// SIMATIC STEP 7 (V5.x) project kuphg_sepGsp2
// CPU: CPU 414-3 PN/DP
// station: P_ADR_BUS
// station: Hardware
// station: kuphg_sepGsp2
// program: S7 Program(2)

SYMBOL_TABLE
"db_Temp"	DB 1	DB 1
"db_BU"	DB 2	DB 2
"db_PIPE"	DB 3	DB 3
"db_Cmmn"	DB 4	DB 4
"idb_fb_Cnvt_Float1"	DB 5	FB 3
"idb_fb_Cnvt_Com"	DB 6	FB 2
"db_MsgCrane"	DB 7	DB 7
"idb_fb_QueueEx"	DB 8	FB 4
"idb_fb_DownloadSnd"	DB 9	FB 10
"idb_fb_Put"	DB 10	FB 6
"idb_fb_Get"	DB 11	FB 7
"idb_fb_Solver"	DB 12	FB 8
"idb_fb_DataFill"	DB 13	FB 9
"db_FIFO"	DB 14	DB 14
"idb_fb_Restart"	DB 15	FB 11
"idb_fb_Scada_Snd"	DB 16	FB 12
"db_MsgInd"	DB 17	DB 17
"idb_fb_Cnvt_Float2"	DB 18	FB 5
"idb_fb_Cnvt_Byte1"	DB 19	FB 14
"idb_fb_Cnvt_Bool1"	DB 20	FB 15
"idb_fb_Cnvt_Bool2"	DB 21	FB 16
"idb_fb_confDown"	DB 22	FB 13
"idb_fb_Snd_Rcv_CP00"	DB 25	FB 18
"idb_fb_Snd_Rcv_CP01"	DB 26	FB 19
"idb_FB_Test"	DB 30	FB 1
"db_MsgCru"	DB 36	DB 36
"idb_fb_StatusRcv"	DB 38	FB 26
"db_MsgPress"	DB 39	DB 39
"db_MsgPPress"	DB 40	DB 40
"db_MsgTemp"	DB 41	DB 41
"db_MsgFlow"	DB 42	DB 42
"db_MsgWorkReg"	DB 43	DB 43
"db_MsgPipeMsg"	DB 44	DB 44
"db_MsgOper"	DB 45	DB 45
"db_MsgInfo"	DB 46	DB 46
"db_MsgOther"	DB 47	DB 47
"idb_snd00"	DB 112	SFB 12
"idb_rcv00"	DB 113	SFB 13
"idb_snd01"	DB 122	SFB 12
"idb_rcv01"	DB 123	SFB 13
"idb_sts00"	DB 201	SFB 22
"idb_sts01"	DB 202	SFB 22
"DbDeb1"	DB 220	DB 220
"DbInfo"	DB 221	DB 221
"DbSensBool"	DB 222	DB 222
"DbSensAI"	DB 223	DB 223
"DbKranPpuAdr"	DB 224	DB 224
"DbKranPpu"	DB 225	DB 225
"DbSepBu"	DB 226	DB 226
"DbSipValve"	DB 227	DB 227
"DbFlowData"	DB 228	DB 228
"DbBitMess"	DB 229	DB 229
"DbControl"	DB 230	DB 230
"DbFlowControl"	DB 231	DB 231
"DbSepBlow"	DB 232	DB 232
"DbCaution"	DB 233	DB 233
"DbEnum"	DB 234	DB 234
"DbSipValveDeb"	DB 248	DB 248
"DbKranPpuDeb"	DB 249	DB 249
"idb_fb_ParScan"	DB 251	FB 251
"idb_fb_KranPpu"	DB 252	FB 252
"idb_fb_Watch"	DB 253	FB 253
"idb_fb_ExecCmd"	DB 254	FB 254
"idb_fb_SipValve"	DB 255	FB 255
"idb_fb_Flow"	DB 256	FB 256
"db_BSEND"	DB 292	SFB 12
"db_BRCV"	DB 293	SFB 13
"DbCpBufSend"	DB 294	DB 294
"DbCpBufRcv"	DB 295	DB 295
"fb_Test"	FB 1	FB 1
"fb_Cnvt_Com"	FB 2	FB 2
"fb_Cnvt_Float1"	FB 3	FB 3
"fb_QueueEx"	FB 4	FB 4
"fb_Cnvt_Float2"	FB 5	FB 5
"fb_Put"	FB 6	FB 6
"fb_Get"	FB 7	FB 7
"fb_Solver"	FB 8	FB 8
"fb_DataFill"	FB 9	FB 9
"fb_DownloadSnd"	FB 10	FB 10
"fb_Restart"	FB 11	FB 11
"fb_Scada_Snd"	FB 12	FB 12
"fb_confDown"	FB 13	FB 13
"fb_Cnvt_Byte1"	FB 14	FB 14
"fb_Cnvt_Bool1"	FB 15	FB 15
"fb_Cnvt_Bool2"	FB 16	FB 16
"fb_Snd_Rcv_CP00"	FB 18	FB 18
"fb_Snd_Rcv_CP01"	FB 19	FB 19
"fb_StatusRcv"	FB 26	FB 26
"fb_ParScan"	FB 251	FB 251
"fb_KranPpu"	FB 252	FB 252
"fb_Watch"	FB 253	FB 253
"fb_ExecCmd"	FB 254	FB 254
"fb_SipValve"	FB 255	FB 255
"fb_Flow"	FB 256	FB 256
"fc_is_empty"	FC 1	FC 1
"CONCAT"	FC 2	FC 2	// Concatenate  String
"fc_MsgSet"	FC 5	FC 5
"fc_MsgReset"	FC 6	FC 6
"fc_MsgHandlerCycle"	FC 7	FC 7
"DT to TOD"	FC 8	FC 8	// DT to TOD
"fc_MsgIsSet"	FC 9	FC 9
"fc_MsgHandlerCrane"	FC 10	FC 10
"I_STRNG"	FC 16	FC 16	// Integer to String
"LEN"	FC 21	FC 21	// Length of String
"MID"	FC 26	FC 26	// Middle Part of String
"RIGHT"	FC 32	FC 32	// Right Part of String
"S5TI_TIM"	FC 33	FC 33	// S5 Time to IEC Time
"SB_DT_DT"	FC 34	FC 34	// Subtract DT - DT
"SB_DT_TM"	FC 35	FC 35	// Subtract DT Time
"TIM_S5TI"	FC 40	FC 40	// IEC Time to S5 Time
"SCALE"	FC 105	FC 105	// Scaling Values
"UNSCALE"	FC 106	FC 106	// Unscaling Values
"FcSetBit"	FC 251	FC 251
"FcBcdByteToInt"	FC 252	FC 252
"FcIntToDt"	FC 253	FC 253
"FcDtToInt"	FC 254	FC 254
"FcDtIntToStr"	FC 255	FC 255
"FcCalcFlow"	FC 256	FC 256
"FcSetCaution"	FC 257	FC 257
"FcPlayCaution"	FC 258	FC 258
"fc_CRC16"	FC 1002	FC 1002	// у Чернова был Fc2 - заменено 20.05.2014
"obMain"	OB 1	OB 1
"obCyclicCalcFlow"	OB 32	OB 32
"obErrRunTime"	OB 80	OB 80
"obRestart"	OB 100	OB 100
"BSEND"	SFB 12	SFB 12	// Sending Segmented Data
"BRCV"	SFB 13	SFB 13	// Receiving Segmented Data
"STATUS"	SFB 22	SFB 22	// Query the Status of a Remote Partner
"SET_CLK"	SFC 0	SFC 0	// Set System Clock
"READ_CLK"	SFC 1	SFC 1	// Read System Clock
"ALARM_SQ"	SFC 17	SFC 17	// Generate Block-Related Messages with Acknowledgment
"ALARM_S"	SFC 18	SFC 18	// Generate Permanently Acknowledged Block-Related Messages
"ALARM_SC"	SFC 19	SFC 19	// Query the Acknowledgment Status of the last ALARM_SQ Entering State Message
"udt_Pipe"	UDT 1	UDT 1
"udt_Pipe_snd"	UDT 4	UDT 4
"udt_Snd"	UDT 5	UDT 5
"udt_Rcv"	UDT 6	UDT 6
"TAdrIOSignal"	UDT 201	UDT 201
"TSignalBool"	UDT 202	UDT 202
"TSignalAI"	UDT 203	UDT 203
"TKranPpu"	UDT 204	UDT 204
"TSepBuParam"	UDT 206	UDT 206
"TSipValve"	UDT 207	UDT 207
"TFlowData"	UDT 208	UDT 208
"TDateTimeBcd"	UDT 209	UDT 209
"TDateTimeInt"	UDT 210	UDT 210
"TSepBlow"	UDT 211	UDT 211
"TCaution"	UDT 212	UDT 212
"TSipValveDeb"	UDT 248	UDT 248
"TKranPpuDeb"	UDT 259	UDT 259
"Vat_Deb_Calc"	VAT 1	
"Vat_AI16_slot10_Piw"	VAT 2	
"Vat_AO8_slot11"	VAT 3	
"Vat_KrPpu_Tmp"	VAT 4	
"Vat_Zagaz"	VAT 5	
"Vat_KrPpu_01_All"	VAT 6	
"Vat_Timer"	VAT 7	
"Vat_DI_09-13zagaz"	VAT 8	
"Vat_Bu_Cfg"	VAT 9	
"Vat_DbSepBu"	VAT 10	
"Vat_Timer_v2"	VAT 11	
"Vat_KlapanSP"	VAT 12	
"Vat_TestBU"	VAT 13	
"vt_dwnld"	VAT 14	
"vt_Message"	VAT 15	
"vt_messtest"	VAT 16	
"vt_msg"	VAT 17	
"vt_Pipe_R0"	VAT 18	
"vt_Pipe_R1"	VAT 19	
"vt_Pipe_R12"	VAT 20	
"vt_Pipe_R6"	VAT 21	
"vt_Pipe_W"	VAT 22	
"vt_queue_ex"	VAT 23	
"vt_snd_rcv"	VAT 24	
"vt_test"	VAT 25	
"Vat_KrPpu_Emul_Si1"	VAT 26	
"Vat_KrPpu_01_Timers"	VAT 27	
"Vat_SensAI_15_Sp_Level"	VAT 28	
"Vat_KrPpu_HandPush"	VAT 29	
"Vat_SensAI_14_Sp_Rashod"	VAT 30	
"Vat_SipValve_3_SP"	VAT 31	
"Vat_KrPpu_All_State_ok"	VAT 32	
"Vat_SipValve_1_Si1"	VAT 33	
"Vat_SipValve_Time"	VAT 34	
"Vat_SipValve_2_Si2"	VAT 35	
"Vat_SipValve_4-5"	VAT 36	
"Vat_Mess"	VAT 37	
"Vat_Emul_Ai_KrPpu_SipVal"	VAT 38	
"Vat_FlowData_0"	VAT 39	
"Vat_FlowControl"	VAT 40	
"Vat_FlowData_1_Gaz_Si1"	VAT 41	
"Vat_ZagazUpr"	VAT 42	
"Vat_BcdDateTime"	VAT 43	
"Vat_FlowData_3_Sp"	VAT 44	
"Vat_BcdDateTime_2"	VAT 45	
"Vat_SensBool_Zagaz"	VAT 46	
"Vat_SensBool2"	VAT 47	
"Vat_SensAI_mA_All"	VAT 48	
"Vat_FlowCalcW"	VAT 49	
"Vat_BU_Uou_KK1"	VAT 50	
"Vat_SensAI_00"	VAT 51	
"Vat_FlowCalcW_1_Si1"	VAT 52	
"Vat_SipValve_4-5a"	VAT 53	
"Vat_FlowCalcW_3_Sp1+"	VAT 54	
"Vat_Caution_tStamp"	VAT 55	
END_SYMBOL_TABLE

TYPE "udt_Pipe"	// UDT 1
VERSION : 0.0
  STRUCT
   CP : INT ;
   PORT : INT ;
   BU : INT ;
   ADDR : BYTE ;	//краны 1,8,11 состояния
   Crane : ARRAY  [0 .. 2 ] OF STRUCT
    Inv : BOOL ;
    RMCntr : BOOL ;
    RComm_Fault : BOOL ;
    RCntr_State : BYTE ;
    RState : BYTE ;
    RCntr_Open : BYTE ;
    RCntr_Close : BYTE ;
    RHw_Error : BYTE ;	//CntrEnableOpen  :BOOL:=0; //0 - нет доступа
//CntrEnableClose  :BOOL:=0; //0 - не
    NeisprUpr : BOOL ;	//0 - неисправность отсутствует
   END_STRUCT ;	//КРУ
   KRU : STRUCT
    Inv : BOOL ;
    RComm_Fault : BOOL ;
    RHw_Fault : BOOL ;
    RCntr_Curr : BOOL ;
    ROpen_Fault : BOOL ;
    RClose_Fault : BOOL ;
    RCntr_Switch : BOOL ;
    RCntr_State : BYTE ;
    RPos_Drv : BYTE ;
    RCntr_Open : BYTE ;
    RCntr_Close : BYTE ;
    RCntr_Pow : BYTE ;
    RCal_Pos_Drv : REAL ;
    RMContr : REAL ;
    RACntr : REAL ;
    RCurr : REAL ;
    RP_PID : REAL ;
    RI_PID : REAL ;
    RD_PID : REAL ;
    CntrEnable : BOOL ;	//0 - нет доступа
    NeisprNoUpr : BOOL ;	//0 - неисправность отсутствует
    NeisprUpr : BOOL ;	//0 - неисправность отсутствует
   END_STRUCT ;
   Press : STRUCT
    Inv : BOOL ;
    RWarnNE : BOOL ;
    RBigNE : BOOL ;
    RWr : BOOL ;
    RA : BYTE ;
    RF : BYTE ;
    RVal : REAL ;
    RUpThres : REAL ;
    RDnThres : REAL ;
    RUpYellow : REAL ;
    RDnYellow : REAL ;
    RUpRed : REAL ;
    RDnRed : REAL ;
    Delta : INT ;
    Zones : INT ;
   END_STRUCT ;
   PPress : STRUCT
    Inv : BOOL ;
    RWr : BOOL ;
    RA : BYTE ;
    RF : BYTE ;
    RVal : REAL ;
    RUpThres : REAL ;
    RDnThres : REAL ;
    RUpYellow : REAL ;
    RDnYellow : REAL ;
    RUpRed : REAL ;
    RDnRed : REAL ;
    Delta : INT ;
    Zones : INT ;
   END_STRUCT ;
   Temp : STRUCT
    Inv : BOOL ;
    RWr : BOOL ;
    RA : BYTE ;
    RF : BYTE ;
    RVal : REAL ;
    RUpThres : REAL ;
    RDnThres : REAL ;
    RUpYellow : REAL ;
    RDnYellow : REAL ;
    RUpRed : REAL ;
    RDnRed : REAL ;
    Delta : INT ;
    Zones : INT ;
   END_STRUCT ;
   POST : STRUCT
    RReq : BOOL ;
    RVal : BOOL ;
   END_STRUCT ;
   FLOW : STRUCT
    Inv : BOOL ;
    RSwitch : BOOL ;
    RWr : BOOL ;
    RFault : BOOL ;
    RVal : REAL ;
    RUst : REAL ;
    RDens : REAL ;
    RDiamDiaf : REAL ;
    RDiamIT : REAL ;
    REqvSh : REAL ;
    RPressBar : REAL ;
    RCo2 : REAL ;
    RNitro : REAL ;
    RRad : REAL ;
    RCnt : REAL ;
    RFlowHour : REAL ;
    RFlowDay : REAL ;
    bSetpoint : BOOL ;
    bSetCalc : BOOL ;
    bSetHBD : BOOL ;
    bSetDBD : BOOL ;
    currHcalc : REAL ;
    prevHcalc : REAL ;
    currDcalc : REAL ;
    prevDcalc : REAL ;
    deltaFlow : REAL ;
    RiseFlow : REAL ;
   END_STRUCT ;
   WrkRegim : STRUCT
    RSwRegWrk : BOOL ;
    RGRP : BOOL ;
    RCntrReg : BYTE ;
    RRegWrk : BYTE ;
   END_STRUCT ;
   PipeMess : STRUCT
    RAlarmRed : BOOL ;
    RFaultTehn : BOOL ;
    RFaultCntr : BOOL ;
    RFaultHW : BOOL ;
    RFaultInt : BOOL ;
    RPermAlarm : BOOL ;
    RRstIntFault : BOOL ;
    RRepair : BOOL ;
    RGasNotBleed : BOOL ;
    RPipeGas : BOOL ;
   END_STRUCT ;
   Times : STRUCT
    RTime : ARRAY  [0 .. 10 ] OF BYTE ;
    RYear : INT ;
    RMonth : INT ;
    RDay : INT ;
    RDay_of_Week : INT ;
    RHour : INT ;
    RMinute : INT ;
    RSecond : INT ;
    RMSecond : INT ;
   END_STRUCT ;
   Ind : INT ;
   Invalid : BOOL ;
   CntrEnable : BOOL ;
   PipeWrkRegim : INT ;
   PipeSeason : INT ;
   cntrIOCranes : BOOL ;
   cntrCCrane : BOOL ;
   inCcIOCranes : BOOL ;
   inCcCCrane : BOOL ;
   inPmaxEkm : BOOL ;
   inPminEkm : BOOL ;
   cntrLedCCraneOP : BOOL ;
   inCCraneOP : BOOL ;
   inCcPmaxEkm : BOOL ;
   inCcPminEkm : BOOL ;
   bAlarmStopWinCC : BOOL ;
  END_STRUCT ;	
END_TYPE

TYPE "udt_Pipe_snd"	// UDT 4
VERSION : 0.0
  STRUCT 	//краны 1,8,11
   Crane : ARRAY  [0 .. 2 ] OF STRUCT
    WMCntr : BOOL ;
   END_STRUCT ;	//КРУ
   KRU : STRUCT
    WCntr_Switch : BOOL ;
    WMContr : REAL ;
    WP_PID : REAL ;
    WI_PID : REAL ;
    WD_PID : REAL ;
   END_STRUCT ;
   Press : STRUCT
    WWr : BOOL ;
    WUpThres : REAL ;
    WDnThres : REAL ;
    WUpYellow : REAL ;
    WDnYellow : REAL ;
    WUpRed : REAL ;
    WDnRed : REAL ;
   END_STRUCT ;
   PPress : STRUCT
    WWr : BOOL ;
    WUpThres : REAL ;
    WDnThres : REAL ;
    WUpYellow : REAL ;
    WDnYellow : REAL ;
    WUpRed : REAL ;
    WDnRed : REAL ;
   END_STRUCT ;
   Temp : STRUCT
    WWr : BOOL ;
    WUpThres : REAL ;
    WDnThres : REAL ;
    WUpYellow : REAL ;
    WDnYellow : REAL ;
    WUpRed : REAL ;
    WDnRed : REAL ;
   END_STRUCT ;
   POST : STRUCT
    WVal : BOOL ;
   END_STRUCT ;
   FLOW : STRUCT
    WSwitch : BOOL ;
    WWr : BOOL ;
    WUst : REAL ;
    WDens : REAL ;
    WDiamDiaf : REAL ;
    WDiamIT : REAL ;
    WEqvSh : REAL ;
    WPressBar : REAL ;
    WCo2 : REAL ;
    WNitro : REAL ;
    WRad : REAL ;
   END_STRUCT ;
   WrkRegim : STRUCT
    WSwRegWrk : BOOL ;
    WGRP : BOOL ;
    WCntrReg : BYTE ;
   END_STRUCT ;
   PipeMess : STRUCT
    WPermAlarm : BOOL ;
    WRstIntFault : BOOL ;
   END_STRUCT ;
   Times : STRUCT
    WTime : ARRAY  [0 .. 10 ] OF BYTE ;
    WYear : INT ;
    WMonth : INT ;
    WDay : INT ;
    WDay_of_Week : INT ;
    WHour : INT ;
    WMinute : INT ;
    WSecond : INT ;
    WMSecond : INT ;
   END_STRUCT ;
  END_STRUCT ;	
END_TYPE

TYPE "udt_Snd"	// UDT 5
VERSION : 0.0
  STRUCT
   adress : BYTE ;
   funct : BYTE ;
   Reg : WORD ;
   Ndata : INT ;
   Data : ARRAY  [0 .. 126 ] OF WORD ;
   Lenght : WORD ;
   Cmd : INT ;	// 0-опрос, 1-команда, 2-загрузка
   Pipe_N : INT ;
   Obj_N : INT ;
   Par_N : INT ;
   Bit : INT ;
  END_STRUCT ;	
END_TYPE

TYPE "udt_Rcv"	// UDT 6
VERSION : 0.0
  STRUCT
   rcv : ARRAY  [0 .. 126 ] OF WORD ;
   Ready : BOOL ;
   Invalid : BOOL ;
  END_STRUCT ;	
END_TYPE

TYPE "TAdrIOSignal"	// UDT 201
VERSION : 0.0
  STRUCT
   adr1 : INT ;
   adr2 : INT ;
  END_STRUCT ;	
END_TYPE

TYPE "TSignalBool"	// UDT 202
VERSION : 0.0
  STRUCT
   adr1 : INT ;
   adr2 : INT ;
   Value : BOOL ;
  END_STRUCT ;	
END_TYPE

TYPE "TSignalAI"	// UDT 203
VERSION : 0.0
  STRUCT
   adrPIW : INT ;	//адрес "слова" в PIW[] для вычисления значения датчика на AI-входе
   ValueIn : INT ;	//пре-обработанное цифровое значение датчика
   Value_mA : REAL ;	//токовое значение датчика (в мА)
   tStamp : DATE_AND_TIME ;	//метка времени в момент успешной обработки значения AI-датчика
   Value : REAL ;	//значение датчиков в момент tStamp (напр. +25.7 градС)
   Value_Subst : REAL ;	//+подстановочное значение
   SubstIncrement : REAL ;	//+ежецикличное приращение для подстановочного значения (меняет знак)
   lblErr : INT ;	//Признак ошибки:0-нет\1-отриц. переполн(<3.8мА)\2-переполн(>20.2мА)\3-обрыв
   lblBound : INT ;	//Признак наруш. границ:-1-неопр\0-Норма\1-LoLo\2-Lo\3-Hi\4-HiHi\>4-ошЗадГраниц
   lblModeSubst : BOOL ;	//+метка активации режима "подстановка значения": 1- "подстановка" \0-нет
   lblModeRepair : BOOL ;	//+метка активации режима "датчик в ремонте" : 1- "в ремонте" \0-нет
   lblSubstCalc : BOOL ;	//+метка активации "простого" пересчёта Value_Subst: 1- пересчитывать \0-нет
   lblSubstCalcBlow : BOOL ;	//+метка активации пересчёта Value_Subst с учетом продувок : 1- да\0-нет
   BoundLoLo : REAL ;	//нижняя аварийная граница
   BoundLo : REAL ;	//нижняя предупредительная граница
   BoundHi : REAL ;	//верхняя предупредительная граница
   BoundHiHi : REAL ;	//верхняя аварийная граница
   LoMeasure : REAL ;	//нижний предел измерения в физич. единицах (напр. -50 градС)
   HiMeasure : REAL ;	//верхний предел измерения в физич. единицах(напр. +100 градС)
   LoMeasure_mA : REAL ;	//нижний предел измерения,мА (const 4 мА для датчиков [4-20]мА)
   HiMeasure_mA : REAL ;	//верхний предел измерения,мА (const 20 мА для датчиков [4-20]мА)
   LoWorkRange_mA : REAL ;	//нижний рабочий предел измерения,мА (напр. 3.8 мА для датчиков [4-20]мА)
   HiWorkRange_mA : REAL ;	//верхний рабочий предел измерения,мА (напр. 20.2 мА для датчиков [4-20]мА)
   HmiBoundLoLo : REAL ;	//дублирующий пакет уставок для независимой корректировки на ВУ
   HmiBoundLo : REAL ;
   HmiBoundHi : REAL ;
   HmiBoundHiHi : REAL ;
   HmiLoMeasure : REAL ;
   HmiHiMeasure : REAL ;
   HmiLoWorkRange_mA : REAL ;
   HmiHiWorkRange_mA : REAL ;
   HmiSyncRange : INT ;	//синхр-ция знач. уставок ПЛК и ВУ:0-не проводить\1-синхрПЛК=>ВУ\2-синхрВУ=>ПЛК
   HmiSensAiDefect : BOOL ;	// Признак ошибочных показаний датчика для ВУ : 0 - правильные \ 1 - ошибочные
  END_STRUCT ;	
END_TYPE

TYPE "TKranPpu"	// UDT 204
VERSION : 0.0
  STRUCT
   KrClose : BOOL ;	//значение DI-сигнала крана ЭППУ "закрыт" (концевик закрытия)
   KrOpen : BOOL ;	//значение DI-сигнала крана ЭППУ "открыт" (концевик открытия)
   CC_Close : BOOL ;	//значение DI-сигнала крана ЭППУ "Целостность Цепи закрытия" :1 - естьЦЦ\0-нет
   CC_Open : BOOL ;	//значение DI-сигнала крана ЭППУ "Целостность Цепи открытия" :1 - естьЦЦ\0-нет
   KrToCloseR : BOOL ;	//значение DO-сигнала крана ЭППУ "закрыть" (чтение состояния)
   KrToCloseW : BOOL ;	//значение DO-сигнала "закрыть" (вычисляется за цикл и назначается в Q[x,5])
   KrToOpenR : BOOL ;	//значение DO-сигнала крана ЭППУ "открыть" (чтение состояния)
   KrToOpenW : BOOL ;	//значение DO-сигнала "открыть" (вычисляется за цикл и назначается в Q[x,5])
   KrToCloseW_HandPush : BOOL ;	//значение DO-сигнала "закрыть" (назначается в Q[x,5] при HandPush=true)
   KrToOpenW_HandPush : BOOL ;	//значение DO-сигнала "открыть" (назначается в Q[x,6] при HandPush=true)
   KrClose_NotSancMove : BOOL ;	//метка : 1- начало несанкцинир. закрытия крана с площадки \ 0- нет)
   KrOpen_NotSancMove : BOOL ;	//метка : 1- начало несанкцинир. открытия крана с площадки \ 0- нет)
   KrClose_PrevVal : BOOL ;	//предыдущее значение DI-сигнала крана ЭППУ "закрыт" (концевик закрытия)
   KrClose_Ev01 : BOOL ;	//флаг события "концевик закрытия замкнулся" (0->1) : 1- да \ 0- нет)
   KrClose_Ev10 : BOOL ;	//флаг события "концевик закрытия разомкнулся" (1->0) : 1- да \ 0- нет)
   KrOpen_PrevVal : BOOL ;	//предыдущее значение DI-сигнала крана ЭППУ "открыт" (концевик открытия)
   KrOpen_Ev01 : BOOL ;	//флаг события "концевик открытия замкнулся" (0->1) : 1- да \ 0- нет)
   KrOpen_Ev10 : BOOL ;	//флаг события "концевик открытия разомкнулся" (1->0) : 1- да \ 0- нет)
   TmOperKr_NO : INT ;	//номер таймера (используютя глобально) - инициализируется
   TmOperKr_TV : S5TIME ;	//величина таймера (длительность) - назначается взавис. от шага операции
   TmOperKr_Q : BOOL ;	//состояние таймера (для таймера типа s_odts : 1 - время отсчитано)
   TmStrag_Value : S5TIME ;	//время на страгивани крана
   TmFullClose_Value : S5TIME ;	//время на полное закрытие крана
   TmFullOpen_Value : S5TIME ;	//время на полное открытие крана
   TmDogim_Value : S5TIME ;	//время на дожим крана  //s5t#20ms
   HmiTmStrag_Value : DINT ;	//время на страгивани крана - для ВУ тип dInt
   HmiTmFullClose_Value : DINT ;	//время на полное закрытие крана - для ВУ тип dInt
   HmiTmFullOpen_Value : DINT ;	//время на полное открытие крана - для ВУ тип dInt
   HmiTmDogim_Value : DINT ;	//время на дожим крана  //s5t#20ms - для ВУ тип dInt
   State : INT ;	//сост-е крана:0-неопред.\1-закрыт\2-открыт\3-закрывается\4-открывается\5-неиспр
   StateByClOp : INT ;	//сост. крана по концевикам : 1-закрыт\2-открыт\3-ClOp00 (разомкнуты)\4-ClOp11
   CmdKrPpu : INT ;	//команда для крана : 0-нет\1-закрыть (с ВУ) \ 2-открыть (с ВУ)\..
   CmdKrPpuModeExec : INT ;	//режим исп.команды: 0-норм.\1-прин.прерыв.\2-прин.исп\3-экстренное исп.
   CmdKrPpu_Next : INT ;	//следующая команда для крана : 0-нет\1-закрыть (с ВУ) \ 2-открыть (с ВУ)\..
   CmdKrPpuModeExec_Next : INT ;	//режим исп.след.команды: 0-норм.\1-прин.прерыв.\2-прин.исп\3-экстренное исп.
   CmdKrPpuLegal : BOOL ;	//непротиворечивость команды : 0-нельзя исполнять\1-можно исполнять
   CmdKrPpuHandPush : BOOL ;	//ручное директивное управленне : 0-выключено\1-включено
   Oper : INT ;	//вып-яемая операция с краном : 0 - нет операций (стоит)\1-закрыть\2-открыть
   OperStep : INT ;	//шаг вып-яемой операции:0-нет\ 1Х-закрытие(11страг\12fullOpen\13дожим)\ 2Х-откр.
   OperErrorLbl : BOOL ;	//наличие ошибки при выполнении операции с краном : 0 - нет \ 1 - есть
   OperErrorNum : INT ;	//номер ошибки при выполнении операции с краном : 0 - нет ошибок \ 1 ..
   HmiErrCC_Close : BOOL ;	//метка : 1- нарушена ц.ц. на закрытие \ 0- нет
   HmiErrCC_Open : BOOL ;	//метка : 1- нарушена ц.ц. на открытие \ 0- нет
   HmiErrClOp00 : BOOL ;	//метка : 1- оба концевика в 0 (разомкнуты) \ 0- нет (ClOp - Close-Open)
   HmiErrClOp11 : BOOL ;	//метка : 1- оба концевика в 1 (замкнуты) \ 0- нет
   HmiErrMessConfirm : BOOL ;	//метка : 1- не квитированы сообщения \ 0- нет
   HmiSyncTimers : INT ;	//синхр-ция знач. таймеров ПЛК и ВУ:0-не проводить\1-синхрПЛК=>ВУ\2-синхрВУ=>ПЛК
   KrDefectFatal : BOOL ;	//фатальная неисправность крана - управление невозможно
   KrDefectNote : BOOL ;	//предупр. неисправность крана, при которой управление возможно
   HmiKrEnableToClose : BOOL ;	//доступность крана для закрытия с ВУ : 0-не доступен \ 1 - доступен
   HmiKrEnableToOpen : BOOL ;	//доступность крана для открытия с ВУ : 0-не доступен \ 1 - доступен
   HmiKrToClose : BOOL ;	//факт подачи команды на закрытие крана с ВУ : 0- не подана \ 1 - подана
   HmiKrToOpen : BOOL ;	//факт подачи команды на открытие крана с ВУ : 0- не подана \ 1 - подана
   isBan_AutoControl : BOOL ;	//флаг запрета автоматического управления краном: 0-нет запрета\ 1- запрещено
   isBan_HandControl : BOOL ;	//флаг запрета ручного управления краном: 0-нет запрета\ 1- запрещено
   reasonBan_AutoControl : INT ;	//причина запрета автоматического управления краном (RBC_ из DbEnum)
   reasonBan_HandControl : INT ;	//причина запрета ручного управления краном (RBC_ из DbEnum)
  END_STRUCT ;	
END_TYPE

TYPE "TSepBuParam"	// UDT 206
VERSION : 0.0
  STRUCT
   addr : BYTE ;	// дрес блока управления в HEX (из db_BU)
   vDbBu_Pipe0 : INT ;	// номер 1-й нитки для шлейфа 57 БУ (номер эл-та в db_Pipe (начинается с 0)
   vDbBu_Pipe1 : INT ;	// номер 2-й нитки для шлейфа 3 БУ (="db_BU".CP[0].PORT[0-1].BU[0-1].PIPE[1])
   Temp_RVal : REAL ;	// Т - температура газа на 1-й нитке
   Press_RVal : REAL ;	// P - давление газа на 1-й нитке
   PPress_RVal : REAL ;	// dP - перепад давления газа на 1-й нитке
   Flow_RVal : REAL ;	// расход газа на 1-й нитке : мгновенный
   Flow_RFlowHour : REAL ;	// расход газа на 1-й нитке :  за предыдущий час
   Flow_RFlowDay : REAL ;	// расход газа на 1-й нитке :  за сутки
   Flow_RCnt : REAL ;	// расход газа на 1-й нитке : за сезон
   CheckRefresh : REAL ;	// значение сканируемого на обновление параметра (периодическое чтение)
   lblErrDataRefresh : BOOL ;	// Признак ошибки обновления данных в db_Pipe: 0-обновляются \1- не обновляются
   lblCopyErrToInvalid : BOOL ;	// Признак назначения db_PIPE.Invalid=1 при lblErr..=1 : 0-нет\1-копировать
   lblSetSubstValue : BOOL ;	// Признак переназначения "999.9" в параметры db_PIPE : 0-нет \ 1-переназначать
   EmulBuParam : BOOL ;	//*эмуляция параметров из БУ : 0 - выключена (реальные сигпалы!)\ 1 - эмуляция
  END_STRUCT ;	
END_TYPE

TYPE "TSipValve"	// UDT 207
VERSION : 0.0
  STRUCT
   AddrPQW : INT ;	//адрес реального выхода PQW[] для выходного AO-сигнала клапана Sipart
   EmulPQW : BOOL ;	//эмуляция сигналов PQW:0-выключена (реальные сигналы!)\1- эмуляция
   TypeNormClOp : BOOL ;	//тип клапана: 0- нормально закрытый\ 1- нормально открытый
   SignalClOpW : BOOL ;	//значение DO-сигнала "закрыть" : 0-закрыть клапан\ 1- открыть
   SignalClOpW_Prev : BOOL ;	//предыд. значение DO-сигнала SignalClOpW
   ControlModeAuto : BOOL ;	//метка: 1-автоматич. режим упр. клапаном \ 0- ручной
   ControlModeAuto_Prev : BOOL ;	//предыд. значение Sprt_Sp_VentMode_Auto
   ControlModeAuto_ChEnable : BOOL ;	//метка: 1-разрешать автоматический режим\ 0-нет (для огр. [4,5] с ВУ)
   SignalClOpW_EvClose : BOOL ;	//флаг события : подача команды "закрыть клапан"
   SignalClOpW_EvOpen : BOOL ;	//флаг события : подача команды "открыть клапан"
   Value_Task_Percent : INT ;	//заданный процент открытия клапана (]0,100])
   Value_Task_Percent_Prev : INT ;	//предыд. значение процента открытия клапана (]0,100])
   Value_DigitPQW : INT ;	//посланное на PQW цифровое значение [0-27648] (что "висит" на PQW[])
   Value_DigitPQW_Prev : INT ;	//предыд. цифровое значение [0-27648], посланное на PQW
   isBan_AutoControl : BOOL ;	//флаг запрета автоматического управления клапаном: 0-нет запрета\ 1- запрещено
   isBan_HandControl : BOOL ;	//флаг запрета ручного управления клапаном: 0-нет запрета\ 1- запрещено
   reasonBan_AutoControl : INT ;	//причина запрета автоматического управления клапаном (RBC_ из DbEnum)
   reasonBan_HandControl : INT ;	//причина запрета ручного управления клапаном (RBC_ из DbEnum)
  END_STRUCT ;	
END_TYPE

TYPE "TFlowData"	// UDT 208
VERSION : 0.0
  STRUCT
   lblCalcFlow : BOOL ;	//признак: рассчитывать расход по параметру : 1-да \0-нет
   Reset_Data : BOOL ;	//обнуление (инициализация) всех данных по параметру: 1-да \0-нет
   Reset_Count_All : BOOL ;	//сброс всех счётчиков по параметру : 1-да \ 0-нет
   Reset_Count_Hour : BOOL ;	//сброс счётчика за текущий час: 1-да \ 0-нет
   Reset_Count_Day : BOOL ;	//сброс счётчика за текущие сутки : 1-да \ 0-нет
   Reset_Count_Month : BOOL ;	//сброс счётчика за текущий месяц : 1-да \ 0-нет
   Reset_Count_Test : BOOL ;	//сброс счётчика за текущий тест (замер) : 1-да \ 0-нет
   Reset_Count_Season : BOOL ;	//сброс счётчика за сезон : 1-да \ 0-нет
   Test_TimeStart : DATE_AND_TIME ;	//метка времени в момент начала теста (замера)
   Test_TimeEnd : DATE_AND_TIME ;	//метка времени в момент окончания теста
   Test_Start : BOOL ;	//сигнал о моменте начала теста : 1-тест начат \ 0-нет
   Test_End : BOOL ;	//сигнал о моменте окончания теста : 1-тест окончен \ 0-нет
   Test_GoOn : BOOL ;	//+флаг : режим теста включен (тест продолжается): 1-тест включен\ 0-нет
   ni1 : INT ;
   ni2 : INT ;
   ni3 : INT ;
   ni4 : INT ;
   ni5 : INT ;
   ni6 : INT ;
   ni7 : INT ;
   ni8 : INT ;
   ni9 : INT ;
   Flow_Instant_Current : REAL ;	//текущий мгновенный
   Flow_Instant_Prev : REAL ;	//предыдущий мгновенный (для алгоритма)
   Flow_Hour_Current : REAL ;	//за текущий час
   Flow_Hour_Prev : REAL ;	//за предыдущий час
   Flow_Day_Current : REAL ;	//за текущие сутки
   Flow_Day_Prev : REAL ;	//за предыдущие сутки
   Flow_Month_Current : REAL ;	//за текущий месяц
   Flow_Month_Prev : REAL ;	//за предыдущий месяц
   Flow_Test_Current : REAL ;	//за текущий тест (замер)
   Flow_Test_Prev : REAL ;	//за предыдущий тест (замер)
   Flow_Season : REAL ;	//за сезон
   Flow_Season_BU : REAL ;	//за сезон из БУ для справки
   Flow_Hour_Arc : ARRAY  [1 .. 48 ] OF REAL ;	//архив часовых значений (24/48)
   Flow_Day_Arc : ARRAY  [1 .. 31 ] OF REAL ;	//архив суточных значений (31/62)
   Flow_Month_Arc : ARRAY  [1 .. 12 ] OF REAL ;	//архив месячных значений (12/24)
  END_STRUCT ;	
END_TYPE

TYPE "TDateTimeBcd"	// UDT 209
VERSION : 0.0
  STRUCT
   Year : BYTE ;	//год (-2000 (две последние цифры) : 2014г=14(int)=20(byte)
   Month : BYTE ;	//месяц [1-12]
   Day : BYTE ;	//день [1-31]
   Hour : BYTE ;	//час [0-23]
   Minute : BYTE ;	//минута [0-59]
   Sec : BYTE ;	//секунда [0-59]
   MSec1 : BYTE ;	//Миллисекунды (2 старших разряда) [00-99] (24(int) для 245мсек)
   MSec2 : BYTE ;	//[0-3]bit-день недели [1-7]\ [4-7]bit-Миллисек, "единицы" [0-9] (5(int))
  END_STRUCT ;	
END_TYPE

TYPE "TDateTimeInt"	// UDT 210
VERSION : 0.0
  STRUCT
   Year : INT ;	//год (-2000 (две последние цифры) : 2014г=14(int)=20(byte)
   Month : INT ;	//месяц [1-12]
   Day : INT ;	//день [1-31]
   Hour : INT ;	//час [0-23]
   Minute : INT ;	//минута [0-59]
   Sec : INT ;	//секунда [0-59]
   MSec : INT ;	//Миллисекунды [0-999]
  END_STRUCT ;	
END_TYPE

TYPE "TSepBlow"	// UDT 211
VERSION : 0.0
  STRUCT
   BlowState : INT ;	//состояние продувки: 0-Неопр \1-начата (включена) \2-выключена \3-окончена
   ControlObject : INT ;	//чем управлять: 1- клапаном или 2- краном ЭПУУ
   WaterLevel_LoControl : REAL ;	//нижний предел уровня жидкости регулирования в физич. ед.
   WaterLevel_HiControl : REAL ;	//верхний предел регулирования в физич. ед.
   WaterLevel_Value : REAL ;	//=уровень жидкости текущий (дубль датчика Уровня Жидкости)
   BlowTimeDurationMax : INT ;	//max продолжительность продувки (сек)
   BlowTimeIntervalMax : INT ;	//max интервал между продувками (сек)
   BlowCountAll : INT ;	//общее количество продувок клапана (автоматических и ручных)
   BlowCountAuto : INT ;	//количество автоматических продувок клапана
   BlowCountTo0 : BOOL ;	//метка: 1 - сброс количества продувок клапана до 0
   BlowTypeAuto : BOOL ;	//тип текущей продувки: 1- автоматическая \0- ручная
   BlowMessStart : BOOL ;	//метка для сообщения: 1-продувка начата\0-сброс сообщения
   BlowMessEnd : BOOL ;	//метка для сообщения: 1-продувка окончена\0-сброс сообщения
   BlowMessDurationMax : BOOL ;	//метка для сообщения: 1-завершение по max дл-ти\0-сброс сообщения
   BlowTimeStart : DATE_AND_TIME ;	//метка времени в момент начала продувки клапана
   BlowTimeEnd : DATE_AND_TIME ;	//метка времени в момент окончания продувки клапана
   BlowTimeInterval : TIME ;	//интервал между последней и предпоследней продувками
   BlowTimeDuration : TIME ;	//длительность последней продувки клапана
   HmiBlowTimeDuration : REAL ;	//продолжительность продувки для ВУ (сек)
   HmiBlowTimeDuration_Prev : REAL ;	//продолжительность предыдущей продувки (сек)
   HmiBlowTimeInterval : REAL ;	//интервал между проувками для ВУ (сек)
   HmiBlowTimeInterval_Prev : REAL ;	//интервал между проувками предыдущий (сек)
   BlowState_Prev : INT ;	//сост. продувки на предыд. цикле : 0-Неопр \1-начата \2-выключена \3-окончена
   Flow_Instant_Current : REAL ;	//==текущий мгновенный РЖ (дубль датчика РЖ)
   Flow_Instant_Prev : REAL ;	//предыдущий мгновенный РЖ (для алгоритма)
   Flow_Blow_Current : REAL ;	//РЖ за текущую продувку
   Flow_Blow_Prew : REAL ;	//РЖ за предыдущую продувку
   Flow_Post_FullClose : REAL ;	//РЖ в интервале между продувками после "доЗакрытия" клапана
   Flow_Post_FullClose_Prev : REAL ;	//РЖ в интервале между продувками после "доЗакрытия" клапана
   Flow_Sens_Correct_Cut : REAL ;	//!!"отсечка" dX показания датчика РЖ (при V<dX, принимается V=0)
   Flow_Sens_Correct_0 : REAL ;	//!!"смещение нуля" dY показания датчика РЖ (при V>dX, принимается V=V-dY)
   BlowDuration_EvOver : BOOL ;	//!флаг : превышена max длительность продувки
   BlowInterval_EvLessMin : BOOL ;	//!флаг : "частые" продувки (интервал с предыдущей меньше min)
   BlowInterval_EvOver : BOOL ;	//!@@флаг : превышен max интервал между продувками
   ForceClose : BOOL ;	//!@@флаг принудительного закрытия продувки : 1-закрыть\0-нет
   ForceOpen : BOOL ;	//!@@флаг принудительного открытия продувки : 1-открыть\0-нет
   WaterLevel_FixAtOpen : REAL ;	//!значение уровня жидкости в начале продувки (при открытии клапана)
   WaterLevel_FixAtClose : REAL ;	//!значение уровня жидкости в конце продувки (при закрытии клапана)
   Tm_Valve_FullClose : INT ;	//время на "доЗакрытие" клапана (задаётся пользователем)
   ni11 : INT ;
   ni12 : INT ;
   ni13 : INT ;
   ni14 : INT ;
   ni15 : INT ;
   ni16 : INT ;
   ni17 : INT ;
   ni18 : INT ;	// $-Клапан (все Sipart) / #-Продувка (только клапаны на сепараторах) / % - РЖ
   ni19 : INT ;	// % - вычисление РЖ Расхода Жидкости (и управление продувкаим)
   ni20 : INT ;	//ё - было ранее в TSipValve () / ! - изменено в охот(к)у
  END_STRUCT ;	
END_TYPE

TYPE "TCaution"	// UDT 212
VERSION : 0.0
  STRUCT
   Melody : INT ;	// мелодия ("гребёнка") для тревоги
   PlayOn_SepSignal_Svet1 : BOOL ;	// проигрывать тревогу на "Световая синализация: Сепараторы_Порог1"
   PlayOn_SepSignal_Svet2 : BOOL ;	// проигрывать тревогу на "Световая синализация: Сепараторы_Порог2"
   PlayOn_SepSignal_Zvuk1 : BOOL ;	// проигрывать тревогу на "Звуковая синализация: Сепараторы_Порог1"
   PlayOn_OperSignal_Svet : BOOL ;	// проигрывать тревогу на "Световая синализация: Операторная"
   PlayOn_OperSignal_Zvuk : BOOL ;	// проигрывать тревогу на "Звуковая синализация: Операторная"
   PlayOn_UouSignal_Svet : BOOL ;	// проигрывать тревогу на "Световая синализация: УОУ"
  END_STRUCT ;	
END_TYPE

TYPE "TSipValveDeb"	// UDT 248
VERSION : 0.0
  STRUCT
   isBan_AutoControl : BOOL ;	//флаг запрета автоматического управления клапаном: 0-нет запрета\ 1- запрещено
   isBan_HandControl : BOOL ;	//флаг запрета ручного управления клапаном: 0-нет запрета\ 1- запрещено
   reasonBan_AutoControl : INT ;	//причина запрета автоматического управления клапаном (RBC_ из DbEnum)
   reasonBan_HandControl : INT ;	//причина запрета ручного управления клапаном (RBC_ из DbEnum)
  END_STRUCT ;	
END_TYPE

TYPE UDT 249
VERSION : 0.0
  STRUCT
   isBan_AutoControl : BOOL ;	//флаг запрета автоматического управления клапаном: 0-нет запрета\ 1- запрещено
   isBan_HandControl : BOOL ;	//флаг запрета ручного управления клапаном: 0-нет запрета\ 1- запрещено
   reasonBan_AutoControl : INT ;	//причина запрета автоматического управления клапаном (RBC_ из DbEnum)
   reasonBan_HandControl : INT ;	//причина запрета ручного управления клапаном (RBC_ из DbEnum)
  END_STRUCT ;	
END_TYPE

FUNCTION_BLOCK "fb_Test"	// FB 1
VERSION : 0.0
VAR_INPUT
  Mess1 { S7_server := 'alarm_archiv'; S7_a_type := 'alarm_s' }: DWORD ;
  Mess2 { S7_server := 'alarm_archiv'; S7_a_type := 'alarm_s' }: DWORD ;
  Mess3 { S7_server := 'alarm_archiv'; S7_a_type := 'alarm_s' }: DWORD ;
END_VAR
VAR
  go_p : BOOL ;
  go_g : BOOL ;
  go_e : BOOL ;
  empty : BOOL ;
  m_start : BOOL ;
  m_stop : BOOL ;
  ack : BOOL ;
  stat : BOOL ;
  ret : INT ;
  A : ARRAY  [0 .. 2 ] OF REAL  := 1.100000e+000, 2.200000e+000, 3.300000e+000;
  A1 : ARRAY  [0 .. 9 ] OF CHAR ;
  A2 : STRING  [10 ] := '1234567890';
  A3 : ARRAY  [0 .. 2 ] OF REAL  := 2.110000e+001, 2.220000e+001, 2.330000e+001;
  m1 : DWORD ;
  m2 : DWORD ;
  m3 : DWORD ;
  tmpW : INT ;
  i : INT ;
  tmpA : INT ;
  pm : INT ;
  n : INT ;
  ndword : INT ;
  nbit : INT ;
  dw : DWORD ;
  nbitHigh : INT ;
  nbitLow : INT ;
  dwMsg : ARRAY  [0 .. 7 ] OF DWORD ;
  b : BOOL ;
END_VAR
BEGIN
// body was compiled from an SCL source; compiled code not shown
END_FUNCTION_BLOCK

FUNCTION_BLOCK "fb_Cnvt_Com"	// FB 2
VERSION : 0.0
VAR_INPUT
  CP : INT ;
  PORT : INT ;
  BU : INT ;
END_VAR
VAR_TEMP
  i : INT ;
  cnt : INT ;
  max_tmp : REAL ;
  min_tmp : REAL ;
END_VAR
BEGIN
// body was compiled from an SCL source; compiled code not shown
END_FUNCTION_BLOCK

FUNCTION_BLOCK "fb_Cnvt_Float1"	// FB 3
VERSION : 0.0
VAR
  tmp : INT ;
  a : REAL ;
  tmp1 : DWORD ;
  tmp2 : DWORD ;
END_VAR
VAR_TEMP
  i : INT ;
  j : INT ;
  k : INT ;
END_VAR
BEGIN
// body was compiled from an SCL source; compiled code not shown
END_FUNCTION_BLOCK

FUNCTION_BLOCK "fb_QueueEx"	// FB 4
VERSION : 0.0
VAR
  PORT : INT ;
  _PORT : INT ;
  CP : INT ;
  done : ARRAY  [0 .. 1, 0 .. 1 ] OF BOOL ;
  bsnd : ARRAY  [0 .. 1, 0 .. 1 ] OF BOOL ;
  DoneSts : ARRAY  [0 .. 1, 0 .. 1 ] OF BOOL ;
  cnt : ARRAY  [0 .. 1, 0 .. 1 ] OF INT ;
  old_cnt : ARRAY  [0 .. 1, 0 .. 1 ] OF INT ;
  cnt_e : ARRAY  [0 .. 1, 0 .. 1 ] OF INT  := 3, 3, 3, 3;
  s_e : ARRAY  [0 .. 1, 0 .. 1 ] OF INT ;
  s_d : ARRAY  [0 .. 1, 0 .. 1 ] OF INT ;
  _local : ARRAY  [0 .. 1, 0 .. 1, 1 .. 16 ] OF BYTE ;
  clk : ARRAY  [0 .. 1, 0 .. 1 ] OF DINT ;
  clk_out : ARRAY  [0 .. 1, 0 .. 1 ] OF INT ;
  clk_tod_old : ARRAY  [0 .. 1, 0 .. 1 ] OF TIME_OF_DAY ;
  clk_tod : ARRAY  [0 .. 1, 0 .. 1 ] OF TIME_OF_DAY ;
  _clk_dt : ARRAY  [0 .. 1, 0 .. 1 ] OF DATE_AND_TIME ;
  snd_tmp : ARRAY  [0 .. 1, 0 .. 1 ] OF STRUCT
   adress : BYTE ;
   funct : BYTE ;
   Reg : WORD ;
   Ndata : INT ;
   Data : ARRAY  [0 .. 126 ] OF WORD ;
   Lenght : WORD ;
   Cmd : INT ;	// 0-опрос, 1-команда, 2-загрузка
   Pipe_N : INT ;
   Obj_N : INT ;
   Par_N : INT ;
   Bit : INT ;
  END_STRUCT ;
  RcvBuff : ARRAY  [0 .. 1, 0 .. 1 ] OF STRUCT
   rcv : ARRAY  [0 .. 126 ] OF WORD ;
   Ready : BOOL ;
   Invalid : BOOL ;
  END_STRUCT ;
  wlen : ARRAY  [0 .. 1, 0 .. 1 ] OF WORD ;
  Stop_Snd : ARRAY  [0 .. 1, 0 .. 1 ] OF BOOL ;
  go : ARRAY  [0 .. 1, 0 .. 1 ] OF BOOL ;
END_VAR
VAR_TEMP
  i : INT ;
END_VAR
BEGIN
// body was compiled from an SCL source; compiled code not shown
END_FUNCTION_BLOCK

FUNCTION_BLOCK "fb_Cnvt_Float2"	// FB 5
VERSION : 0.0
VAR_TEMP
  i : INT ;
  j : INT ;
  k : INT ;
  tmp1 : INT ;
  tmp2 : INT ;
  tmp3 : INT ;
  tmp4 : INT ;
END_VAR
BEGIN
// body was compiled from an SCL source; compiled code not shown
END_FUNCTION_BLOCK

FUNCTION_BLOCK "fb_Put"	// FB 6
VERSION : 0.0
VAR_INPUT
  CP : INT ;
  Port : INT ;
  snd : STRUCT
   adress : BYTE ;
   funct : BYTE ;
   Reg : WORD ;
   Ndata : INT ;
   Data : ARRAY  [0 .. 126 ] OF WORD ;
   Lenght : WORD ;
   Cmd : INT ;	// 0-опрос, 1-команда, 2-загрузка
   Pipe_N : INT ;
   Obj_N : INT ;
   Par_N : INT ;
   Bit : INT ;
  END_STRUCT ;
END_VAR
VAR_OUTPUT
  Of_err : BOOL ;
END_VAR
BEGIN
// body was compiled from an SCL source; compiled code not shown
END_FUNCTION_BLOCK

FUNCTION_BLOCK "fb_Get"	// FB 7
VERSION : 0.0
VAR_INPUT
  CP : INT ;
  Port : INT ;
END_VAR
VAR_OUTPUT
  snd : STRUCT
   adress : BYTE ;
   funct : BYTE ;
   Reg : WORD ;
   Ndata : INT ;
   Data : ARRAY  [0 .. 126 ] OF WORD ;
   Lenght : WORD ;
   Cmd : INT ;	// 0-опрос, 1-команда, 2-загрузка
   Pipe_N : INT ;
   Obj_N : INT ;
   Par_N : INT ;
   Bit : INT ;
  END_STRUCT ;
  Of_err : BOOL ;
END_VAR
VAR_TEMP
  i : INT ;
END_VAR
BEGIN
// body was compiled from an SCL source; compiled code not shown
END_FUNCTION_BLOCK

FUNCTION_BLOCK "fb_Solver"	// FB 8
VERSION : 0.0
VAR_INPUT
  cnt : INT ;
  CP : INT ;
  PORT : INT ;
  e_cnt : INT ;
  Stop_Snd : ARRAY  [0 .. 1, 0 .. 1 ] OF BOOL ;
END_VAR
VAR_OUTPUT
  snd : ARRAY  [0 .. 1, 0 .. 1 ] OF STRUCT
   adress : BYTE ;
   funct : BYTE ;
   Reg : WORD ;
   Ndata : INT ;
   Data : ARRAY  [0 .. 126 ] OF WORD ;
   Lenght : WORD ;
   Cmd : INT ;	// 0-опрос, 1-команда, 2-загрузка
   Pipe_N : INT ;
   Obj_N : INT ;
   Par_N : INT ;
   Bit : INT ;
  END_STRUCT ;
  cnt_out : ARRAY  [0 .. 1, 0 .. 1 ] OF INT ;
  next : ARRAY  [0 .. 1, 0 .. 1 ] OF BOOL ;
END_VAR
VAR
  cnt_t : ARRAY  [0 .. 1, 0 .. 1, 0 .. 2 ] OF INT  := 0;
  cnt_r : ARRAY  [0 .. 1, 0 .. 1 ] OF INT ;
  snd_dummy : STRUCT
   adress : BYTE ;
   funct : BYTE ;
   Reg : WORD ;
   Ndata : INT ;
   Data : ARRAY  [0 .. 126 ] OF WORD ;
   Lenght : WORD ;
   Cmd : INT ;	// 0-опрос, 1-команда, 2-загрузка
   Pipe_N : INT ;
   Obj_N : INT ;
   Par_N : INT ;
   Bit : INT ;
  END_STRUCT ;
  BU1 : INT ;
  BU2 : INT ;
  download : BOOL ;
  nPipe : INT ;
END_VAR
VAR_TEMP
  i : INT ;
END_VAR
BEGIN
// body was compiled from an SCL source; compiled code not shown
END_FUNCTION_BLOCK

FUNCTION_BLOCK "fb_DataFill"	// FB 9
VERSION : 0.0
VAR_TEMP
  i : INT ;
  j : INT ;
  k : INT ;
END_VAR
BEGIN
// body was compiled from an SCL source; compiled code not shown
END_FUNCTION_BLOCK

FUNCTION_BLOCK "fb_DownloadSnd"	// FB 10
VERSION : 0.0
VAR_INPUT
  cnt_in : INT ;
  CP : INT ;
  PORT : INT ;
  BU : INT ;
END_VAR
VAR_OUTPUT
  snd : ARRAY  [0 .. 1, 0 .. 1 ] OF STRUCT
   adress : BYTE ;
   funct : BYTE ;
   Reg : WORD ;
   Ndata : INT ;
   Data : ARRAY  [0 .. 126 ] OF WORD ;
   Lenght : WORD ;
   Cmd : INT ;	// 0-опрос, 1-команда, 2-загрузка
   Pipe_N : INT ;
   Obj_N : INT ;
   Par_N : INT ;
   Bit : INT ;
  END_STRUCT ;
  cnt_out : ARRAY  [0 .. 1, 0 .. 1 ] OF INT ;
  Busy : ARRAY  [0 .. 1, 0 .. 1, 0 .. 2 ] OF BOOL ;
END_VAR
VAR
  InitCRC : WORD  := W#16#FFFF;
  CRC : ARRAY  [0 .. 1, 0 .. 1, 0 .. 2 ] OF WORD ;
  in : ARRAY  [0 .. 1, 0 .. 1, 0 .. 2, 0 .. 2 ] OF BOOL ;
  out : ARRAY  [0 .. 1, 0 .. 1, 0 .. 2, 0 .. 2 ] OF BOOL ;
  CT : ARRAY  [0 .. 1, 0 .. 1, 0 .. 2, 0 .. 2 ] OF S5TIME ;
  cnt_buff : ARRAY  [0 .. 1, 0 .. 1, 0 .. 2 ] OF INT ;
  dwnl_sucsess : ARRAY  [0 .. 1, 0 .. 1, 0 .. 2 ] OF BOOL ;
END_VAR
VAR_TEMP
  tmp_dw : DWORD ;
  i : INT ;
  j : INT ;
  tmp_len : INT ;
END_VAR
BEGIN
// body was compiled from an SCL source; compiled code not shown
END_FUNCTION_BLOCK

FUNCTION_BLOCK "fb_Restart"	// FB 11
VERSION : 0.0
VAR_TEMP
  i : INT ;
END_VAR
BEGIN
// body was compiled from an SCL source; compiled code not shown
END_FUNCTION_BLOCK

FUNCTION_BLOCK "fb_Scada_Snd"	// FB 12
VERSION : 0.0
VAR
  Pipe_N : INT ;
  Obj_N : INT ;
  Par_N : INT ;
  snd : STRUCT
   adress : BYTE ;
   funct : BYTE ;
   Reg : WORD ;
   Ndata : INT ;
   Data : ARRAY  [0 .. 126 ] OF WORD ;
   Lenght : WORD ;
   Cmd : INT ;	// 0-опрос, 1-команда, 2-загрузка
   Pipe_N : INT ;
   Obj_N : INT ;
   Par_N : INT ;
   Bit : INT ;
  END_STRUCT ;
  bsnd : BOOL ;
  tmp : BOOL ;
  Data : ARRAY  [0 .. 126 ] OF WORD ;
  itmp1 : INT ;
  itmp2 : INT ;
  itmp3 : INT ;
  itmp4 : INT ;
  it1 : INT ;
  it2 : INT ;
  tmp1 : WORD ;
  tmp2 : WORD ;
  tmp3 : WORD ;
  tmp4 : WORD ;
END_VAR
VAR_TEMP
  funct : BYTE ;
  ndata : DINT ;
  Reg : ARRAY  [0 .. 1 ] OF INT ;
  Post : BOOL ;
  Bit : INT ;
  Float : BOOL ;
  Lenght : WORD ;
END_VAR
BEGIN
// body was compiled from an SCL source; compiled code not shown
END_FUNCTION_BLOCK

FUNCTION_BLOCK "fb_confDown"	// FB 13
VERSION : 0.0
VAR_INPUT
  nIn : INT ;
  CP : INT ;
  PORT : INT ;
  BU : INT ;
  nPipe : INT ;
END_VAR
VAR_OUTPUT
  snd : ARRAY  [0 .. 1, 0 .. 1 ] OF STRUCT
   adress : BYTE ;
   funct : BYTE ;
   Reg : WORD ;
   Ndata : INT ;
   Data : ARRAY  [0 .. 126 ] OF WORD ;
   Lenght : WORD ;
   Cmd : INT ;	// 0-опрос, 1-команда, 2-загрузка
   Pipe_N : INT ;
   Obj_N : INT ;
   Par_N : INT ;
   Bit : INT ;
  END_STRUCT ;
  nOut : INT ;
END_VAR
VAR
  InitCRC : WORD  := W#16#FFFF;
  CRC : WORD ;
  nBuff : INT ;
  dwnl_sucsess : BOOL ;
  dwnl_flength : DWORD ;
  tmpFLen : DINT ;
  dwnl_data_cnt : INT ;
  dwnl_data : ARRAY  [0 .. 9 ] OF STRUCT
   data : ARRAY  [0 .. 126 ] OF //Данные
   WORD ;	//Данные
   Length : INT ;	//Длина
   ready : BOOL ;	//готовность true - готов
  END_STRUCT ;
  inf : STRUCT
   address : WORD ;
   vers : WORD ;
  END_STRUCT ;
  dwnl_End : BOOL ;
END_VAR
VAR_TEMP
  tmp_len : INT ;
  i : INT ;
  j : INT ;
END_VAR
BEGIN
// body was compiled from an SCL source; compiled code not shown
END_FUNCTION_BLOCK

FUNCTION_BLOCK "fb_Cnvt_Byte1"	// FB 14
VERSION : 0.0
VAR_TEMP
  i : INT ;
  j : INT ;
  k : INT ;
END_VAR
BEGIN
// body was compiled from an SCL source; compiled code not shown
END_FUNCTION_BLOCK

FUNCTION_BLOCK "fb_Cnvt_Bool1"	// FB 15
VERSION : 0.0
VAR_TEMP
  i : INT ;
  j : INT ;
  k : INT ;
END_VAR
BEGIN
// body was compiled from an SCL source; compiled code not shown
END_FUNCTION_BLOCK

FUNCTION_BLOCK "fb_Cnvt_Bool2"	// FB 16
VERSION : 0.0
VAR
  CP : INT ;
  PORT : INT ;
  BU : INT ;
  out : BOOL ;
END_VAR
VAR_TEMP
  i : INT ;
  j : INT ;
  k : INT ;
END_VAR
BEGIN
// body was compiled from an SCL source; compiled code not shown
END_FUNCTION_BLOCK

FUNCTION_BLOCK "fb_Snd_Rcv_CP00"	// FB 18
VERSION : 0.0
VAR_INPUT
  SndBuff : STRUCT
   adress : BYTE ;
   funct : BYTE ;
   Reg : WORD ;
   Ndata : INT ;
   Data : ARRAY  [0 .. 126 ] OF WORD ;
   Lenght : WORD ;
   Cmd : INT ;	// 0-опрос, 1-команда, 2-загрузка
   Pipe_N : INT ;
   Obj_N : INT ;
   Par_N : INT ;
   Bit : INT ;
  END_STRUCT ;
END_VAR
VAR
  phys : ARRAY  [1 .. 4 ] OF BYTE ;
  logi : ARRAY  [1 .. 4 ] OF BYTE ;
  local : ARRAY  [1 .. 16 ] OF BYTE ;
END_VAR
BEGIN
// body was compiled from an SCL source; compiled code not shown
END_FUNCTION_BLOCK

FUNCTION_BLOCK "fb_Snd_Rcv_CP01"	// FB 19
VERSION : 0.0
VAR_INPUT
  SndBuff : STRUCT
   adress : BYTE ;
   funct : BYTE ;
   Reg : WORD ;
   Ndata : INT ;
   Data : ARRAY  [0 .. 126 ] OF WORD ;
   Lenght : WORD ;
   Cmd : INT ;	// 0-опрос, 1-команда, 2-загрузка
   Pipe_N : INT ;
   Obj_N : INT ;
   Par_N : INT ;
   Bit : INT ;
  END_STRUCT ;
END_VAR
VAR
  phys : ARRAY  [1 .. 4 ] OF BYTE ;
  logi : ARRAY  [1 .. 4 ] OF BYTE ;
  local : ARRAY  [1 .. 16 ] OF BYTE ;
END_VAR
BEGIN
// body was compiled from an SCL source; compiled code not shown
END_FUNCTION_BLOCK

FUNCTION_BLOCK "fb_StatusRcv"	// FB 26
VERSION : 0.0
VAR_INPUT
  cnt : INT ;
  CP : INT ;
  PORT : INT ;
  DoneSts : BOOL ;
  snd : STRUCT
   adress : BYTE ;
   funct : BYTE ;
   Reg : WORD ;
   Ndata : INT ;
   Data : ARRAY  [0 .. 126 ] OF WORD ;
   Lenght : WORD ;
   Cmd : INT ;	// 0-опрос, 1-команда, 2-загрузка
   Pipe_N : INT ;
   Obj_N : INT ;
   Par_N : INT ;
   Bit : INT ;
  END_STRUCT ;
END_VAR
VAR
  rcv_NULL : STRUCT
   rcv : ARRAY  [0 .. 126 ] OF WORD ;
   Ready : BOOL ;
   Invalid : BOOL ;
  END_STRUCT ;
  cnt_t : INT ;
  dwnl_sucsess : ARRAY  [0 .. 1, 0 .. 1, 0 .. 2 ] OF BOOL ;
END_VAR
BEGIN
// body was compiled from an SCL source; compiled code not shown
END_FUNCTION_BLOCK

FUNCTION_BLOCK "fb_ParScan"	// FB 251
TITLE = Циклический опрос параметров
AUTHOR : Konst
FAMILY : Main
NAME : ParScan
VERSION : 1.0
VAR
  Cycle : REAL ;
  Tm1 : S5TIME ;
  Tm1Impuls : BOOL  := TRUE;
  Tm1Value : S5TIME  := S5T#20MS;	//длительность одного кванта времени
  Quant_Tm1 : INT  := 1;	//счетчик квантов времени, отсчитываемых таймером Tm1
  nQuant_Tm1 : INT  := 10;	//число квантов времени, насчитываемых таймером Tm1
  Tm2 : S5TIME ;
  Tm2Impuls : BOOL  := TRUE;
  Tm2Value : S5TIME  := S5T#3S;	//период проверки
  resScale_SensAIParam : WORD ;
  vt1 : REAL ;
  BoundNotControl : REAL  := 8.888880e+002;	//Уставки с таким значением не контролируются
  BoundLbl : INT ;	//промежуточная для вычисления  DbSensAI.SensAIParam[n1].lblBound
  ni_RangeAiNorm : INT  := 27648;
  nr_RangeAiNorm : REAL ;
  SubstErrVal : REAL  := 9.999000e+002;	//Значение для замещения ошибочного значения параметра (исп.для AI-датчиков и в d
END_VAR
VAR_TEMP
  i1 : INT ;
  it1 : INT ;
  j1 : INT ;
  n1 : INT ;
  indP : INT ;
  ndt1 : DATE_AND_TIME ;
  nr1 : REAL ;
  nr2 : REAL ;
  nw1 : WORD ;
END_VAR
BEGIN
// body was compiled from an SCL source; compiled code not shown
END_FUNCTION_BLOCK

FUNCTION_BLOCK "fb_KranPpu"	// FB 252
TITLE = Работа с кранами ЭППУ
AUTHOR : Konst
FAMILY : Main
NAME : ParScan
VERSION : 1.0
VAR
  Cycle : REAL ;
  TmOperStartImpulse : ARRAY  [1 .. 15 ] OF BOOL ;
  TmOperState : ARRAY  [1 .. 15 ] OF INT ;
  TmOperResult : ARRAY  [1 .. 15 ] OF S5TIME ;
  lblDopWork : ARRAY  [1 .. 15 ] OF //1- доп. обработка по крану нужна \ 0 - не нужна
  BOOL ;	//1- доп. обработка по крану нужна \ 0 - не нужна
END_VAR
VAR_TEMP
  nbl1 : BOOL ;
  nbl2 : BOOL ;
  lblOpOk : BOOL ;
  i1 : INT ;
  it1 : INT ;
  ni1 : INT ;
  ndt1 : DATE_AND_TIME ;
END_VAR
BEGIN
// body was compiled from an SCL source; compiled code not shown
END_FUNCTION_BLOCK

FUNCTION_BLOCK "fb_Watch"	// FB 253
TITLE = Наблюдение за состоянием, командами, ошибками
AUTHOR : Konst
FAMILY : Main
NAME : Watch
VERSION : 1.0
VAR
  DoAutoControl : BOOL ;	//true - выполнять алгоритм автоматического управления
  ControlJob : INT ;	//код задания команд по управлению : 0-нет\1-run\2-stop\3-"+5"\4-"-5"
END_VAR
VAR_TEMP
  i1 : INT ;
  j1 : INT ;
  n1 : INT ;
  ni1 : INT ;
  ni2 : INT ;
  ndt1 : DATE_AND_TIME ;
  nr1 : REAL ;
END_VAR
BEGIN
// body was compiled from an SCL source; compiled code not shown
END_FUNCTION_BLOCK

FUNCTION_BLOCK "fb_ExecCmd"	// FB 254
TITLE = Выполнение команд управления
AUTHOR : Konst
FAMILY : Main
NAME : ExecCmd
VERSION : 1.0
VAR
  Cycle : REAL ;
  JobWrPkw : STRUCT
   Write1 : WORD ;
   Write2 : WORD ;
   Write3 : WORD ;
   Write4 : WORD ;
  END_STRUCT ;
  JobWrPzd : STRUCT
   Write1 : WORD ;
   Write2 : WORD ;
  END_STRUCT ;
  lblExecStepCmd : BOOL ;	//true - выполнять очередной шаг CurrentStep \ false - отдых
  w1 : WORD ;
  w2 : WORD ;
  w3 : WORD ;
  w4 : WORD ;
END_VAR
VAR_TEMP
  ni1 : INT ;
  ndt1 : DATE_AND_TIME ;
  nr1 : REAL ;
  nr2 : REAL ;
  nr3 : REAL ;
  nr4 : REAL ;
  wrd3 : WORD ;
  wrd4 : WORD ;
  dwrd1 : DWORD ;
  dwrd2 : DWORD ;
END_VAR
BEGIN
// body was compiled from an SCL source; compiled code not shown
END_FUNCTION_BLOCK

FUNCTION_BLOCK "fb_SipValve"	// FB 255
TITLE = Управление клапанами Sipart
AUTHOR : Konst
FAMILY : Main
NAME : SipValve
VERSION : 1.0
VAR
  Cycle : REAL ;
  TimePlc : DATE_AND_TIME ;	//текущее время ПЛК
  TimePlcSet : BOOL ;
END_VAR
VAR_TEMP
  lblBlowType : BOOL ;
  lblChangeDigitPQW : BOOL ;
  lblChangeMode : BOOL ;
  lblSendControlSignal : BOOL ;
  i1 : INT ;
  n1 : INT ;
  n2 : INT ;
  ni1 : INT ;
  nr1 : REAL ;
  nr2 : REAL ;
  wLevel : REAL ;
  nr_RangeAoNorm : REAL ;
  nr_Percent : REAL ;
  ndt1 : DATE_AND_TIME ;
END_VAR
BEGIN
// body was compiled from an SCL source; compiled code not shown
END_FUNCTION_BLOCK

FUNCTION_BLOCK "fb_Flow"	// FB 256
TITLE = Проведение операций в DbFlowData
AUTHOR : Konst
FAMILY : Main
NAME : Flow
VERSION : 1.0
VAR
  TimePlc : DATE_AND_TIME ;	//текущее время ПЛК
  curMonth : INT ;
  curDay : INT ;
  curHour : INT ;
  td1 : TIME_OF_DAY ;	//TOD
  NullVal : REAL ;	//Значение для )
  NullDebVal : REAL  := 1.200000e+000;	//Значение для )
  DtStr1 : STRING  [22 ];	//TimePlc в строковом виде: "21.05.14 15:25:34.640"
END_VAR
VAR_TEMP
  i1 : INT ;
  j1 : INT ;
  n1 : INT ;
  n2 : INT ;
  ni1 : INT ;
  ni2 : INT ;
  ndt1 : DATE_AND_TIME ;
  ndt2 : DATE_AND_TIME ;
  nr1 : REAL ;
END_VAR
BEGIN
// body was compiled from an SCL source; compiled code not shown
END_FUNCTION_BLOCK

FUNCTION_BLOCK FB 291
TITLE = Разработка1
AUTHOR : Konst
FAMILY : Main
NAME : FbCpExch
VERSION : 1.0
VAR
  countCycle : REAL ;
  dCount : REAL  := 1.000000e-004;	//приращение счетчиков
  BreakCount : BOOL ;	//Назначается True для сброса счетчиков
  StopSend : BOOL ;	//обход вызова BSEND
  Start_Req : BOOL  := TRUE;
  RestartPostOk : BOOL  := TRUE;
  RestartPostErr : BOOL  := TRUE;
  RestartPostReceive : BOOL ;
  NumCpBuf : INT  := 1;
  pS_REQ : BOOL  := TRUE;
  pS_R : BOOL ;
  pS_ID : WORD  := W#16#1010;	//см. в NetPro какой LocalID на конкретном порту CP
  pS_R_ID : DWORD ;
  pS_Len : WORD  := W#16#6;
  pS_DONE : BOOL ;
  pS_ERROR : BOOL ;
  pS_STATUS : WORD ;
  pS_REQ_Prev : BOOL ;
  pS_DONE_Prev : BOOL ;
  pS_ERROR_Prev : BOOL ;
  pS_STATUS_Prev : WORD ;
  pS_REQ_Count : REAL ;
  pS_DONE_Count : REAL ;
  pS_ERROR_Count : REAL ;
  pS_STATUS_Count : REAL ;
  pS_STATUS_PrevNotNull : WORD ;
  StopReceive : BOOL ;
  Start_EN_R : BOOL  := TRUE;
  pR_EN_R : BOOL  := TRUE;
  pR_ID : WORD ;	//:=w#16#1010;   // см. в NetPro какой LocalID на конкретном порту CP
  pR_R_ID : DWORD ;
  pR_Len : WORD ;
  pR_NDR : BOOL ;
  pR_ERROR : BOOL ;
  pR_STATUS : WORD ;
  pR_EN_R_Prev : BOOL ;
  pR_NDR_Prev : BOOL ;
  pR_ERROR_Prev : BOOL ;
  pR_STATUS_Prev : WORD ;
  pR_EN_R_Count : REAL ;
  pR_NDR_Count : REAL ;
  pR_ERROR_Count : REAL ;
  pR_STATUS_Count : REAL ;
  pR_STATUS_PrevNotNull : WORD ;
  pR_Len_PrevNotNull : WORD ;
END_VAR
VAR_TEMP
  rcvSymbol : BYTE ;
  ni1 : INT ;
END_VAR
BEGIN
// body was compiled from an SCL source; compiled code not shown
END_FUNCTION_BLOCK

FUNCTION "fc_is_empty" : BOOL	// FC 1
VERSION : 0.0
VAR_INPUT
  CP : INT ;
  Port : INT ;
END_VAR
VAR_OUTPUT
  RET_VAL : BOOL ;
END_VAR
BEGIN
// body was compiled from an SCL source; compiled code not shown
END_FUNCTION

// FC 2: know-how protected block, not included

FUNCTION "fc_MsgSet" : VOID	// FC 5
VERSION : 0.0
VAR_INPUT
  typ : INT ;
  p : INT ;
  pm : INT ;
  icrane : INT ;
END_VAR
VAR_TEMP
  ndword : INT ;
  nbit : INT ;
  dw : DWORD ;
END_VAR
BEGIN
// body was compiled from an SCL source; compiled code not shown
END_FUNCTION

FUNCTION "fc_MsgReset" : VOID	// FC 6
VERSION : 0.0
VAR_INPUT
  typ : INT ;
  p : INT ;
  pm : INT ;
  icrane : INT ;
END_VAR
VAR_TEMP
  ndword : INT ;
  nbit : INT ;
  dw : DWORD ;
END_VAR
BEGIN
// body was compiled from an SCL source; compiled code not shown
END_FUNCTION

FUNCTION "fc_MsgHandlerCycle" : VOID	// FC 7
VERSION : 0.0
VAR_INPUT
  CP : INT ;
  PORT : INT ;
  BU : INT ;
END_VAR
VAR_TEMP
  i : INT ;
END_VAR
BEGIN
// body was compiled from an SCL source; compiled code not shown
END_FUNCTION

// FC 8: know-how protected block, not included

FUNCTION "fc_MsgIsSet" : BOOL	// FC 9
VERSION : 0.0
VAR_INPUT
  typ : INT ;
  flag_ack : BOOL ;	//flag := 0, ack := 1
  p : INT ;
  pm : INT ;
  icrane : INT ;
END_VAR
VAR_OUTPUT
  RET_VAL : BOOL ;
END_VAR
VAR_TEMP
  ndword : INT ;
  nbit : INT ;
  dw : DWORD ;
END_VAR
BEGIN
// body was compiled from an SCL source; compiled code not shown
END_FUNCTION

FUNCTION "fc_MsgHandlerCrane" : VOID	// FC 10
VERSION : 0.0
VAR_INPUT
  CP : INT ;
  PORT : INT ;
  BU : INT ;
  p : INT ;
END_VAR
VAR_TEMP
  npipe : INT ;
  i : INT ;
END_VAR
BEGIN
// body was compiled from an SCL source; compiled code not shown
END_FUNCTION

// FC 16: know-how protected block, not included

// FC 21: know-how protected block, not included

// FC 26: know-how protected block, not included

// FC 32: know-how protected block, not included

// FC 33: know-how protected block, not included

// FC 34: know-how protected block, not included

// FC 35: know-how protected block, not included

// FC 40: know-how protected block, not included

// FC 105: know-how protected block, not included

// FC 106: know-how protected block, not included

FUNCTION "FcSetBit" : WORD	// FC 251
TITLE = FcSetBit
AUTHOR : Konst
FAMILY : Main
NAME : FcSetBit
VERSION : 1.0
VAR_INPUT
  ObjW : WORD ;
  NumPos : INT ;
  BitVal_W : BOOL ;
END_VAR
VAR_OUTPUT
  RET_VAL : WORD ;
END_VAR
VAR_TEMP
  nbl1 : BOOL ;
  nw1 : WORD ;
  nw2 : WORD ;
  nw3 : WORD ;
END_VAR
BEGIN
// body was compiled from an SCL source; compiled code not shown
END_FUNCTION

FUNCTION "FcBcdByteToInt" : INT	// FC 252
TITLE = BcdByte_ToInt
AUTHOR : Konst
FAMILY : Main
NAME : BcdByte
VERSION : 1.0
VAR_INPUT
  ObjB : BYTE ;
END_VAR
VAR_OUTPUT
  RET_VAL : INT ;
END_VAR
VAR_TEMP
  nbt1 : BYTE ;
  nbt2 : BYTE ;
  ni1 : INT ;
  ni2 : INT ;
END_VAR
BEGIN
// body was compiled from an SCL source; compiled code not shown
END_FUNCTION

FUNCTION "FcIntToDt" : DATE_AND_TIME	// FC 253
TITLE = FcIntToDt
AUTHOR : Konst
FAMILY : Main
NAME : IntToDt
VERSION : 1.0
VAR_INPUT
  ObjDtInt : STRUCT
   Year : INT ;	//год (-2000 (две последние цифры) : 2014г=14(int)=20(byte)
   Month : INT ;	//месяц [1-12]
   Day : INT ;	//день [1-31]
   Hour : INT ;	//час [0-23]
   Minute : INT ;	//минута [0-59]
   Sec : INT ;	//секунда [0-59]
   MSec : INT ;	//Миллисекунды [0-999]
  END_STRUCT ;
END_VAR
VAR_OUTPUT
  RET_VAL : DATE_AND_TIME ;
END_VAR
VAR_TEMP
  ni1 : INT ;
  dtBcd : STRUCT
   Year : BYTE ;	//год (-2000 (две последние цифры) : 2014г=14(int)=20(byte)
   Month : BYTE ;	//месяц [1-12]
   Day : BYTE ;	//день [1-31]
   Hour : BYTE ;	//час [0-23]
   Minute : BYTE ;	//минута [0-59]
   Sec : BYTE ;	//секунда [0-59]
   MSec1 : BYTE ;	//Миллисекунды (2 старших разряда) [00-99] (24(int) для 245мсек)
   MSec2 : BYTE ;	//[0-3]bit-день недели [1-7]\ [4-7]bit-Миллисек, "единицы" [0-9] (5(int))
  END_STRUCT ;
END_VAR
BEGIN
// body was compiled from an SCL source; compiled code not shown
END_FUNCTION

FUNCTION "FcDtToInt" : VOID	// FC 254
TITLE = FcIntToDt
AUTHOR : Konst
FAMILY : Main
NAME : IntToDt
VERSION : 1.0
VAR_INPUT
  ndt1 : DATE_AND_TIME ;
END_VAR
VAR_OUTPUT
  ObjDtInt : STRUCT
   Year : INT ;	//год (-2000 (две последние цифры) : 2014г=14(int)=20(byte)
   Month : INT ;	//месяц [1-12]
   Day : INT ;	//день [1-31]
   Hour : INT ;	//час [0-23]
   Minute : INT ;	//минута [0-59]
   Sec : INT ;	//секунда [0-59]
   MSec : INT ;	//Миллисекунды [0-999]
  END_STRUCT ;
END_VAR
VAR_TEMP
  ni1 : INT ;
  dtBcd : STRUCT
   Year : BYTE ;	//год (-2000 (две последние цифры) : 2014г=14(int)=20(byte)
   Month : BYTE ;	//месяц [1-12]
   Day : BYTE ;	//день [1-31]
   Hour : BYTE ;	//час [0-23]
   Minute : BYTE ;	//минута [0-59]
   Sec : BYTE ;	//секунда [0-59]
   MSec1 : BYTE ;	//Миллисекунды (2 старших разряда) [00-99] (24(int) для 245мсек)
   MSec2 : BYTE ;	//[0-3]bit-день недели [1-7]\ [4-7]bit-Миллисек, "единицы" [0-9] (5(int))
  END_STRUCT ;
END_VAR
BEGIN
// body was compiled from an SCL source; compiled code not shown
END_FUNCTION

FUNCTION "FcDtIntToStr" : STRING	// FC 255
TITLE = FcIntToDt
AUTHOR : Konst
FAMILY : Main
NAME : IntToDt
VERSION : 1.0
VAR_INPUT
  ObjDtInt : STRUCT
   Year : INT ;	//год (-2000 (две последние цифры) : 2014г=14(int)=20(byte)
   Month : INT ;	//месяц [1-12]
   Day : INT ;	//день [1-31]
   Hour : INT ;	//час [0-23]
   Minute : INT ;	//минута [0-59]
   Sec : INT ;	//секунда [0-59]
   MSec : INT ;	//Миллисекунды [0-999]
  END_STRUCT ;
END_VAR
VAR_OUTPUT
  RET_VAL : STRING  [254 ];
END_VAR
VAR_TEMP
  str0 : STRING  [4 ];
  str1 : STRING  [22 ];
  str2 : STRING  [22 ];
END_VAR
BEGIN
// body was compiled from an SCL source; compiled code not shown
END_FUNCTION

FUNCTION "FcCalcFlow" : VOID	// FC 256
TITLE = FcSetBit
AUTHOR : Konst
FAMILY : Main
NAME : FcSetBit
VERSION : 1.0
VAR_TEMP
  lblBlowDuration_EvOver : BOOL ;	//BlowDuration_EvOver lblEvOver
  i1 : INT ;
  n1 : INT ;
  chBlowState_FromTo : INT ;	//изменение BlowState за цикл : 0- нет\12: 1->2 \23: 2->3 \31: 3->1 \21: 2->1 \1(
  calcCycle : REAL ;	//цикл опроса в секундах
  nr1 : REAL ;	//цикл опроса в секундах
  Flow1Cycle : REAL ;	//приращение РЖ за цикл сканирования с учётом погрешности датчика РЖ
  nw1 : WORD ;
END_VAR
BEGIN
// body was compiled from an SCL source; compiled code not shown
END_FUNCTION

FUNCTION "FcSetCaution" : VOID	// FC 257
TITLE = FcSetCaution
AUTHOR : Konst
FAMILY : Main
NAME : FcSetBit
VERSION : 1.0
VAR_INPUT
  CautionID : INT ;
END_VAR
VAR_TEMP
  cID : INT ;
  ni1 : INT ;
  TimePlc : DATE_AND_TIME ;	//текущее время ПЛК
END_VAR
BEGIN
// body was compiled from an SCL source; compiled code not shown
END_FUNCTION

FUNCTION "FcPlayCaution" : VOID	// FC 258
TITLE = FcPlayCaution
AUTHOR : Konst
FAMILY : Main
NAME : FcSetBit
VERSION : 1.0
VAR_TEMP
  nw1 : WORD ;
END_VAR
BEGIN
// body was compiled from an SCL source; compiled code not shown
END_FUNCTION

FUNCTION "fc_CRC16" : WORD	// FC 1002
VERSION : 0.0
VAR_INPUT
  CRC : WORD ;
  length : INT ;
  data : ARRAY  [0 .. 126 ] OF WORD ;
END_VAR
VAR_OUTPUT
  RET_VAL : WORD ;
END_VAR
VAR_TEMP
  i : INT ;
  j : INT ;
  ind : INT ;
  flag : BOOL ;
  tmp : WORD ;
  data_b : ARRAY  [0 .. 254 ] OF BYTE ;
END_VAR
BEGIN
// body was compiled from an SCL source; compiled code not shown
END_FUNCTION

DATA_BLOCK "db_Temp"	// DB 1
//Присвоение переменных
//
VERSION : 0.0
  STRUCT
   Old_P : ARRAY  [0 .. 23 ] OF UDT 1;
  END_STRUCT ;	
BEGIN
END_DATA_BLOCK

DATA_BLOCK "db_BU"	// DB 2
//В Этом блоке описаны переменные связанные с блоками управления, концепция состоит в том что на у контроллера 
//есть два коммуникационных процессора,в каждом коммуникационном
//процессоре есть 2 порта и на каждом порту висят три блока управления. Каждый блок управления обслуживает 2 нитки(шлейфа).
//На нитку приходится две команды опроса параметров 
//Нельзя присваивать разным блокам одинаковые номера ниток
///Количество блоков 12, количество шлейфов 24
//
VERSION : 0.0
  STRUCT
   CP : ARRAY  [0 .. 1 ] OF STRUCT
    PORT : ARRAY  [0 .. 1 ] OF STRUCT
     BU : ARRAY  [0 .. 2 ] OF STRUCT
      Addr : BYTE ;	//Адрес блока управления в HEX
      PIPE : ARRAY  [0 .. 1 ] OF INT ;	//Номера ниток(шлейфов)
      BU_Regim : INT ;	//Режим работы блока управления
      cnt : INT ;
      rcv_tmp : UDT 6;
      snd : ARRAY  [0 .. 1 ] OF UDT 5;	//посылки команд
      rcv : ARRAY  [0 .. 1 ] OF UDT 6;	//буфер приема ответов на команды
      dwnl_End : BOOL ;	//Признак окнчания загрузки true - конец
      dwnl_Sucsess : BOOL ;	//Признак успеха загрузки true - успех
      dwnl_Half_e1 : BOOL ;	//Признак готовности первой половины буфера true - готов
      dwnl_Half_e2 : BOOL ;	//Признак готовности второй половины буфера true - готов
      dwnl_data_cnt : INT ;
      dwnl_flength : DWORD ;	//Длина передаваемого файла в байтах
      dwnl_data : ARRAY  [0 .. 9 ] OF STRUCT 	//Массив структур буферов на передачу
       data : ARRAY  [0 .. 126 ] OF WORD ;	//Данные
       Length : INT ;	//Длина
       ready : BOOL ;	//готовность true - готов
      END_STRUCT ;
     END_STRUCT ;
    END_STRUCT ;
   END_STRUCT ;
  END_STRUCT ;	
BEGIN
   CP[0].PORT[0].BU[0].Addr := B#16#2;
   CP[0].PORT[0].BU[0].PIPE[1] := 10;
   CP[0].PORT[0].BU[0].snd[0].adress := B#16#2;
   CP[0].PORT[0].BU[0].snd[0].funct := B#16#2;
   CP[0].PORT[0].BU[0].snd[0].Reg := W#16#64;
   CP[0].PORT[0].BU[0].snd[0].Ndata := 758;
   CP[0].PORT[0].BU[0].snd[0].Lenght := W#16#6;
   CP[0].PORT[0].BU[0].snd[1].adress := B#16#2;
   CP[0].PORT[0].BU[0].snd[1].funct := B#16#2;
   CP[0].PORT[0].BU[0].snd[1].Reg := W#16#3E8;
   CP[0].PORT[0].BU[0].snd[1].Ndata := 1012;
   CP[0].PORT[0].BU[0].snd[1].Lenght := W#16#6;
   CP[0].PORT[0].BU[1].Addr := B#16#3;
   CP[0].PORT[0].BU[1].PIPE[0] := 1;
   CP[0].PORT[0].BU[1].PIPE[1] := 11;
   CP[0].PORT[0].BU[1].snd[0].adress := B#16#3;
   CP[0].PORT[0].BU[1].snd[0].funct := B#16#2;
   CP[0].PORT[0].BU[1].snd[0].Reg := W#16#64;
   CP[0].PORT[0].BU[1].snd[0].Ndata := 758;
   CP[0].PORT[0].BU[1].snd[0].Lenght := W#16#6;
   CP[0].PORT[0].BU[1].snd[1].adress := B#16#3;
   CP[0].PORT[0].BU[1].snd[1].funct := B#16#2;
   CP[0].PORT[0].BU[1].snd[1].Reg := W#16#3E8;
   CP[0].PORT[0].BU[1].snd[1].Ndata := 1012;
   CP[0].PORT[0].BU[1].snd[1].Lenght := W#16#6;
   CP[0].PORT[0].BU[2].Addr := B#16#22;
   CP[0].PORT[0].BU[2].PIPE[0] := 22;
   CP[0].PORT[0].BU[2].PIPE[1] := 22;
   CP[0].PORT[1].BU[0].Addr := B#16#4;
   CP[0].PORT[1].BU[0].PIPE[0] := 2;
   CP[0].PORT[1].BU[0].PIPE[1] := 12;
   CP[0].PORT[1].BU[0].snd[0].adress := B#16#4;
   CP[0].PORT[1].BU[0].snd[0].funct := B#16#2;
   CP[0].PORT[1].BU[0].snd[0].Reg := W#16#64;
   CP[0].PORT[1].BU[0].snd[0].Ndata := 758;
   CP[0].PORT[1].BU[0].snd[0].Lenght := W#16#6;
   CP[0].PORT[1].BU[0].snd[1].adress := B#16#4;
   CP[0].PORT[1].BU[0].snd[1].funct := B#16#2;
   CP[0].PORT[1].BU[0].snd[1].Reg := W#16#3E8;
   CP[0].PORT[1].BU[0].snd[1].Ndata := 1012;
   CP[0].PORT[1].BU[0].snd[1].Lenght := W#16#6;
   CP[0].PORT[1].BU[1].Addr := B#16#5;
   CP[0].PORT[1].BU[1].PIPE[0] := 3;
   CP[0].PORT[1].BU[1].PIPE[1] := 13;
   CP[0].PORT[1].BU[1].snd[0].adress := B#16#5;
   CP[0].PORT[1].BU[1].snd[0].funct := B#16#2;
   CP[0].PORT[1].BU[1].snd[0].Reg := W#16#64;
   CP[0].PORT[1].BU[1].snd[0].Ndata := 758;
   CP[0].PORT[1].BU[1].snd[0].Lenght := W#16#6;
   CP[0].PORT[1].BU[1].snd[1].adress := B#16#5;
   CP[0].PORT[1].BU[1].snd[1].funct := B#16#2;
   CP[0].PORT[1].BU[1].snd[1].Reg := W#16#3E8;
   CP[0].PORT[1].BU[1].snd[1].Ndata := 1012;
   CP[0].PORT[1].BU[1].snd[1].Lenght := W#16#6;
   CP[0].PORT[1].BU[2].Addr := B#16#22;
   CP[0].PORT[1].BU[2].PIPE[0] := 22;
   CP[0].PORT[1].BU[2].PIPE[1] := 22;
   CP[1].PORT[0].BU[0].Addr := B#16#22;
   CP[1].PORT[0].BU[0].PIPE[0] := 22;
   CP[1].PORT[0].BU[0].PIPE[1] := 22;
   CP[1].PORT[0].BU[1].Addr := B#16#22;
   CP[1].PORT[0].BU[1].PIPE[0] := 22;
   CP[1].PORT[0].BU[1].PIPE[1] := 22;
   CP[1].PORT[0].BU[2].Addr := B#16#22;
   CP[1].PORT[0].BU[2].PIPE[0] := 22;
   CP[1].PORT[0].BU[2].PIPE[1] := 22;
   CP[1].PORT[1].BU[0].Addr := B#16#22;
   CP[1].PORT[1].BU[0].PIPE[0] := 22;
   CP[1].PORT[1].BU[0].PIPE[1] := 22;
   CP[1].PORT[1].BU[1].Addr := B#16#22;
   CP[1].PORT[1].BU[1].PIPE[0] := 22;
   CP[1].PORT[1].BU[1].PIPE[1] := 22;
   CP[1].PORT[1].BU[2].Addr := B#16#22;
   CP[1].PORT[1].BU[2].PIPE[0] := 22;
   CP[1].PORT[1].BU[2].PIPE[1] := 22;
END_DATA_BLOCK

DATA_BLOCK "db_PIPE"	// DB 3
//Присвоение переменных
//
VERSION : 0.0
  STRUCT
   P : ARRAY  [0 .. 23 ] OF UDT 1;
   P_snd : UDT 4;
  END_STRUCT ;	
BEGIN
END_DATA_BLOCK

DATA_BLOCK "db_Cmmn"	// DB 4
//Общие переменные проекта
//
VERSION : 0.0
  STRUCT
   Scd_Send : BOOL ;	//Признак посылки команды со скады  true - признак активен
   BU_recnfg : BOOL ;	//Запрос на изменение конфигурации блоков, ниток true - запрос активен
   GSP_Regim : INT ;	//режим работы ГСП 0-отбор 1- закачка 2-аварийный останов
   Restart_Post : ARRAY  [0 .. 23 ] OF BOOL  := TRUE, TRUE, TRUE, TRUE, TRUE, TRUE, TRUE, TRUE, TRUE, TRUE, TRUE, TRUE, TRUE, TRUE, TRUE, TRUE, TRUE, TRUE, TRUE, TRUE, TRUE, TRUE, TRUE, TRUE;	//Массив начальных состояний ПОСТА
   FirstStartCPU : BOOL ;	// Добавлено 12.11.13 по просьбе ЛещевойИ
   RezhimRabotiGSP : INT ;	// Добавлено 12.11.13 по просьбе ЛещевойИ
  END_STRUCT ;	
BEGIN
   Restart_Post[0] := TRUE;
   Restart_Post[1] := TRUE;
   Restart_Post[2] := TRUE;
   Restart_Post[3] := TRUE;
   Restart_Post[4] := TRUE;
   Restart_Post[5] := TRUE;
   Restart_Post[6] := TRUE;
   Restart_Post[7] := TRUE;
   Restart_Post[8] := TRUE;
   Restart_Post[9] := TRUE;
   Restart_Post[10] := TRUE;
   Restart_Post[11] := TRUE;
   Restart_Post[12] := TRUE;
   Restart_Post[13] := TRUE;
   Restart_Post[14] := TRUE;
   Restart_Post[15] := TRUE;
   Restart_Post[16] := TRUE;
   Restart_Post[17] := TRUE;
   Restart_Post[18] := TRUE;
   Restart_Post[19] := TRUE;
   Restart_Post[20] := TRUE;
   Restart_Post[21] := TRUE;
   Restart_Post[22] := TRUE;
   Restart_Post[23] := TRUE;
END_DATA_BLOCK

DATA_BLOCK "idb_fb_Cnvt_Float1"	// DB 5
VERSION : 0.0
"fb_Cnvt_Float1"
BEGIN
END_DATA_BLOCK

DATA_BLOCK "idb_fb_Cnvt_Com"	// DB 6
VERSION : 0.0
"fb_Cnvt_Com"
BEGIN
END_DATA_BLOCK

DATA_BLOCK "db_MsgCrane"	// DB 7
// nMsg, nPipe, nCrane
//
VERSION : 0.0
  STRUCT
   event : ARRAY  [0 .. 7, 0 .. 23, 0 .. 2 ] OF DWORD ;
   flag : ARRAY  [0 .. 7, 0 .. 23, 0 .. 2 ] OF DWORD ;
   ack : ARRAY  [0 .. 7, 0 .. 23, 0 .. 2 ] OF DWORD ;
  END_STRUCT ;	
BEGIN
END_DATA_BLOCK

DATA_BLOCK "idb_fb_QueueEx"	// DB 8
VERSION : 0.0
"fb_QueueEx"
BEGIN
END_DATA_BLOCK

DATA_BLOCK "idb_fb_DownloadSnd"	// DB 9
VERSION : 0.0
"fb_DownloadSnd"
BEGIN
END_DATA_BLOCK

DATA_BLOCK "idb_fb_Put"	// DB 10
VERSION : 0.0
"fb_Put"
BEGIN
END_DATA_BLOCK

DATA_BLOCK "idb_fb_Get"	// DB 11
VERSION : 0.0
"fb_Get"
BEGIN
END_DATA_BLOCK

DATA_BLOCK "idb_fb_Solver"	// DB 12
VERSION : 0.0
"fb_Solver"
BEGIN
END_DATA_BLOCK

DATA_BLOCK "idb_fb_DataFill"	// DB 13
VERSION : 0.0
"fb_DataFill"
BEGIN
END_DATA_BLOCK

DATA_BLOCK "db_FIFO"	// DB 14
//Данные буфера
//
VERSION : 0.0
  STRUCT
   FIFO : ARRAY  [0 .. 1, 0 .. 1 ] OF STRUCT
    snd : ARRAY  [0 .. 20 ] OF UDT 5;
   END_STRUCT ;
   P_ind : ARRAY  [0 .. 1, 0 .. 1 ] OF INT  := 0, 0, 0, 0;
   G_ind : ARRAY  [0 .. 1, 0 .. 1 ] OF INT  := 0, 0, 0, 0;
   End : INT  := 20;
  END_STRUCT ;	
BEGIN
   End := 20;
END_DATA_BLOCK

DATA_BLOCK "idb_fb_Restart"	// DB 15
VERSION : 0.0
"fb_Restart"
BEGIN
END_DATA_BLOCK

DATA_BLOCK "idb_fb_Scada_Snd"	// DB 16
VERSION : 0.0
"fb_Scada_Snd"
BEGIN
END_DATA_BLOCK

DATA_BLOCK "db_MsgInd"	// DB 17
//nMsgInd, nPipe, nInd
//
VERSION : 0.0
  STRUCT
   i : ARRAY  [0 .. 300, 0 .. 23, 0 .. 1 ] OF REAL ;
  END_STRUCT ;	
BEGIN
END_DATA_BLOCK

DATA_BLOCK "idb_fb_Cnvt_Float2"	// DB 18
VERSION : 0.0
"fb_Cnvt_Float2"
BEGIN
END_DATA_BLOCK

DATA_BLOCK "idb_fb_Cnvt_Byte1"	// DB 19
VERSION : 0.0
"fb_Cnvt_Byte1"
BEGIN
END_DATA_BLOCK

DATA_BLOCK "idb_fb_Cnvt_Bool1"	// DB 20
VERSION : 0.0
"fb_Cnvt_Bool1"
BEGIN
END_DATA_BLOCK

DATA_BLOCK "idb_fb_Cnvt_Bool2"	// DB 21
VERSION : 0.0
"fb_Cnvt_Bool2"
BEGIN
END_DATA_BLOCK

DATA_BLOCK "idb_fb_confDown"	// DB 22
VERSION : 0.0
"fb_confDown"
BEGIN
END_DATA_BLOCK

DATA_BLOCK "idb_fb_Snd_Rcv_CP00"	// DB 25
VERSION : 0.0
"fb_Snd_Rcv_CP00"
BEGIN
END_DATA_BLOCK

DATA_BLOCK "idb_fb_Snd_Rcv_CP01"	// DB 26
VERSION : 0.0
"fb_Snd_Rcv_CP01"
BEGIN
END_DATA_BLOCK

DATA_BLOCK "idb_FB_Test"	// DB 30
VERSION : 0.0
"fb_Test"
BEGIN
END_DATA_BLOCK

DATA_BLOCK "db_MsgCru"	// DB 36
// nMsg, nPipe
//
VERSION : 0.0
  STRUCT
   event : ARRAY  [0 .. 7, 0 .. 23 ] OF DWORD ;
   flag : ARRAY  [0 .. 7, 0 .. 23 ] OF DWORD ;
   ack : ARRAY  [0 .. 7, 0 .. 23 ] OF DWORD ;
  END_STRUCT ;	
BEGIN
END_DATA_BLOCK

DATA_BLOCK "idb_fb_StatusRcv"	// DB 38
VERSION : 0.0
"fb_StatusRcv"
BEGIN
END_DATA_BLOCK

DATA_BLOCK "db_MsgPress"	// DB 39
// nMsg, nPipe
//
VERSION : 0.0
  STRUCT
   event : ARRAY  [0 .. 7, 0 .. 23 ] OF DWORD ;
   flag : ARRAY  [0 .. 7, 0 .. 23 ] OF DWORD ;
   ack : ARRAY  [0 .. 7, 0 .. 23 ] OF DWORD ;
  END_STRUCT ;	
BEGIN
END_DATA_BLOCK

DATA_BLOCK "db_MsgPPress"	// DB 40
// nMsg, nPipe
//
VERSION : 0.0
  STRUCT
   event : ARRAY  [0 .. 7, 0 .. 23 ] OF DWORD ;
   flag : ARRAY  [0 .. 7, 0 .. 23 ] OF DWORD ;
   ack : ARRAY  [0 .. 7, 0 .. 23 ] OF DWORD ;
  END_STRUCT ;	
BEGIN
END_DATA_BLOCK

DATA_BLOCK "db_MsgTemp"	// DB 41
// nMsg, nPipe
//
VERSION : 0.0
  STRUCT
   event : ARRAY  [0 .. 7, 0 .. 23 ] OF DWORD ;
   flag : ARRAY  [0 .. 7, 0 .. 23 ] OF DWORD ;
   ack : ARRAY  [0 .. 7, 0 .. 23 ] OF DWORD ;
  END_STRUCT ;	
BEGIN
END_DATA_BLOCK

DATA_BLOCK "db_MsgFlow"	// DB 42
// nMsg, nPipe
//
VERSION : 0.0
  STRUCT
   event : ARRAY  [0 .. 7, 0 .. 23 ] OF DWORD ;
   flag : ARRAY  [0 .. 7, 0 .. 23 ] OF DWORD ;
   ack : ARRAY  [0 .. 7, 0 .. 23 ] OF DWORD ;
  END_STRUCT ;	
BEGIN
END_DATA_BLOCK

DATA_BLOCK "db_MsgWorkReg"	// DB 43
// nMsg, nPipe
//
VERSION : 0.0
  STRUCT
   event : ARRAY  [0 .. 7, 0 .. 23 ] OF DWORD ;
   flag : ARRAY  [0 .. 7, 0 .. 23 ] OF DWORD ;
   ack : ARRAY  [0 .. 7, 0 .. 23 ] OF DWORD ;
  END_STRUCT ;	
BEGIN
END_DATA_BLOCK

DATA_BLOCK "db_MsgPipeMsg"	// DB 44
// nMsg, nPipe
//
VERSION : 0.0
  STRUCT
   event : ARRAY  [0 .. 7, 0 .. 23 ] OF DWORD ;
   flag : ARRAY  [0 .. 7, 0 .. 23 ] OF DWORD ;
   ack : ARRAY  [0 .. 7, 0 .. 23 ] OF DWORD ;
  END_STRUCT ;	
BEGIN
END_DATA_BLOCK

DATA_BLOCK "db_MsgOper"	// DB 45
// nMsg, nPipe
//
VERSION : 0.0
  STRUCT
   event : ARRAY  [0 .. 16, 0 .. 23 ] OF DWORD ;
   flag : ARRAY  [0 .. 16, 0 .. 23 ] OF DWORD ;
   ack : ARRAY  [0 .. 16, 0 .. 23 ] OF DWORD ;
  END_STRUCT ;	
BEGIN
END_DATA_BLOCK

DATA_BLOCK "db_MsgInfo"	// DB 46
// nMsg, nPipe
//
VERSION : 0.0
  STRUCT
   event : ARRAY  [0 .. 16, 0 .. 23 ] OF DWORD ;
   flag : ARRAY  [0 .. 16, 0 .. 23 ] OF DWORD ;
   ack : ARRAY  [0 .. 16, 0 .. 23 ] OF DWORD ;
  END_STRUCT ;	
BEGIN
END_DATA_BLOCK

DATA_BLOCK "db_MsgOther"	// DB 47
// nMsg, nPipe
//
VERSION : 0.0
  STRUCT
   event : ARRAY  [0 .. 16, 0 .. 23 ] OF DWORD ;
   flag : ARRAY  [0 .. 16, 0 .. 23 ] OF DWORD ;
   ack : ARRAY  [0 .. 16, 0 .. 23 ] OF DWORD ;
  END_STRUCT ;	
BEGIN
END_DATA_BLOCK

DATA_BLOCK "idb_snd00"	// DB 112
AUTHOR : SIMATIC
FAMILY : COM_FUNC
VERSION : 0.0
"BSEND"
BEGIN
END_DATA_BLOCK

DATA_BLOCK "idb_rcv00"	// DB 113
AUTHOR : SIMATIC
FAMILY : COM_FUNC
VERSION : 0.0
"BRCV"
BEGIN
END_DATA_BLOCK

DATA_BLOCK "idb_snd01"	// DB 122
AUTHOR : SIMATIC
FAMILY : COM_FUNC
VERSION : 0.0
"BSEND"
BEGIN
END_DATA_BLOCK

DATA_BLOCK "idb_rcv01"	// DB 123
AUTHOR : SIMATIC
FAMILY : COM_FUNC
VERSION : 0.0
"BRCV"
BEGIN
END_DATA_BLOCK

DATA_BLOCK "idb_sts00"	// DB 201
AUTHOR : SIMATIC
FAMILY : COM_FUNC
VERSION : 0.0
"STATUS"
BEGIN
END_DATA_BLOCK

DATA_BLOCK "idb_sts01"	// DB 202
AUTHOR : SIMATIC
FAMILY : COM_FUNC
VERSION : 0.0
"STATUS"
BEGIN
END_DATA_BLOCK

DATA_BLOCK "DbDeb1"	// DB 220
TITLE = 'Отладка врем.'
AUTHOR : Konst
FAMILY : Deb1
NAME : DbDeb1
VERSION : 0.0
  STRUCT
   tmp1 : ARRAY  [0 .. 1000 ] OF BYTE ;
   nbl1 : BOOL ;
   nbl2 : BOOL ;
   nbl3 : BOOL ;
   nbl4 : BOOL ;
   nbl5 : BOOL ;
   nbl6 : BOOL ;
   nbl7 : BOOL ;
   nbl8 : BOOL ;
   nbl9 : BOOL ;
   nbl10 : BOOL ;
   nbt1 : BYTE ;
   nbt2 : BYTE ;
   nbt3 : BYTE ;
   nbt4 : BYTE ;
   nbt5 : BYTE ;
   nbt6 : BYTE ;
   nbt7 : BYTE ;
   nbt8 : BYTE ;
   nbt9 : BYTE ;
   nbt10 : BYTE ;
   ni1 : INT ;
   ni2 : INT ;
   ni3 : INT ;
   ni4 : INT ;
   ni5 : INT ;
   ni6 : INT ;
   ni7 : INT ;
   ni8 : INT ;
   ni9 : INT ;
   ni10 : INT ;
   nr1 : REAL ;
   nr2 : REAL ;
   nr3 : REAL ;
   nr4 : REAL ;
   nr5 : REAL ;
   nr6 : REAL ;
   nr7 : REAL ;
   nr8 : REAL ;
   nr9 : REAL ;
   nr10 : REAL ;
   nw1 : WORD ;
   nw2 : WORD ;
   nw3 : WORD ;
   nw4 : WORD ;
   nw5 : WORD ;
   nw6 : WORD ;
   nw7 : WORD ;
   nw8 : WORD ;
   nw9 : WORD ;
   nw10 : WORD ;
   nw11 : WORD ;
   nw12 : WORD ;
   nw13 : WORD ;
   nw14 : WORD ;
   nw15 : WORD ;
   nw16 : WORD ;
   nw17 : WORD ;
   nw18 : WORD ;
   nw19 : WORD ;
   nw20 : WORD ;
   nw21 : WORD ;
   nw22 : WORD ;
   nw23 : WORD ;
   nw24 : WORD ;
   nw25 : WORD ;
   nw26 : WORD ;
   nw27 : WORD ;
   nw28 : WORD ;
   nw29 : WORD ;
   nw30 : WORD ;
   ndw1 : DWORD ;
   ndw2 : DWORD ;
   ndw3 : DWORD ;
   ndw4 : DWORD ;
   ndw5 : DWORD ;
   ndw6 : DWORD ;
   ndw7 : DWORD ;
   ndw8 : DWORD ;
   ndw9 : DWORD ;
   ndw10 : DWORD ;
   ns1 : STRING  [250 ];
   ns2 : STRING  [250 ];
   ns3 : STRING  [250 ];
   ns4 : STRING  [250 ];
   ns5 : STRING  [250 ];
   ns6 : STRING  [250 ];
   ns7 : STRING  [250 ];
   ns8 : STRING  [250 ];
   ns9 : STRING  [250 ];
   ns10 : STRING  [250 ];
   ndt1 : DATE_AND_TIME ;
   ndt2 : DATE_AND_TIME ;
   ndt3 : DATE_AND_TIME ;
   ndt4 : DATE_AND_TIME ;
   ndt5 : DATE_AND_TIME ;
   ndt6 : DATE_AND_TIME ;
   ndt7 : DATE_AND_TIME ;
   ndt8 : DATE_AND_TIME ;
   ndt9 : DATE_AND_TIME ;
   ndt10 : DATE_AND_TIME ;
   deb1 : INT ;
   deb2 : INT ;
   deb3 : INT ;
   deb4 : INT ;
   deb5 : INT ;
   deb6 : INT ;
   deb7 : INT ;
   deb8 : INT ;
   deb9 : INT ;
   deb10 : INT ;
   deb11 : INT ;
   deb12 : INT ;
   deb13 : INT ;
   deb14 : INT ;
   deb15 : INT ;
   deb16 : INT ;
   deb17 : INT ;
   deb18 : INT ;
   deb19 : INT ;
   deb20 : INT ;
  END_STRUCT ;	//Db
BEGIN
END_DATA_BLOCK

DATA_BLOCK "DbInfo"	// DB 221
TITLE = 'Общая информация'
AUTHOR : Konst
FAMILY : Main
NAME : DbInfo
VERSION : 0.0
  STRUCT
   Ver : WORD ;
   k1 : INT ;
   k2 : INT ;
   k3 : INT ;
   ExchangeBU : BOOL ;
  END_STRUCT ;	//Db
BEGIN
   ExchangeBU := TRUE;
END_DATA_BLOCK

DATA_BLOCK "DbSensBool"	// DB 222
TITLE = 'Значения параметров '
AUTHOR : Konst
FAMILY : Main
NAME : DbZagaz
VERSION : 0.0
  STRUCT
   numZagazBlockInSep : INT ;
   numZagazBlockInUou : INT ;
   numZagazBlockInOper : INT ;
   ZagazPar_SepBlock : ARRAY  [1 .. 6, 1 .. 2 ] OF UDT 202;
   ZagazPar_OperBlock : ARRAY  [1 .. 1, 1 .. 2 ] OF UDT 202;
   ZagazPar_UouBlock : ARRAY  [1 .. 10, 1 .. 2 ] OF UDT 202;
   ZagazPar_SepCHM10 : UDT 202;
   ZagazPar_UouCHM10 : UDT 202;
   PtnPar_HeaterOn : UDT 202;
   PtnPar_HeaterBreak : UDT 202;
   PtnPar_P_malo : UDT 202;
   VsbPar_P_DoE1Malo : UDT 202;
   VsbPar_P_PosleE1Malo : UDT 202;
   LitPar_T_ObrVodii_AvtVkl : UDT 202;
   LitPar_ObogrevIT_Vkl : UDT 202;
   LitPar_ObogrevIT_Viikl : UDT 202;
   LitPar_ObogrevIT_Avariia : UDT 202;
   ZagazUpr_SepSignal_Svet1 : UDT 202;
   ZagazUpr_SepSignal_Svet2 : UDT 202;
   ZagazUpr_SepSignal_Zvuk1 : UDT 202;
   ZagazUpr_OperSignal_Svet : UDT 202;
   ZagazUpr_OperSignal_Zvuk : UDT 202;
   ZagazUpr_UouSignal_Svet : UDT 202;
  END_STRUCT ;	//Db
BEGIN
   numZagazBlockInSep := 6;
   numZagazBlockInUou := 10;
   numZagazBlockInOper := 1;
   ZagazPar_SepBlock[1, 1].adr1 := 12;
   ZagazPar_SepBlock[1, 2].adr1 := 12;
   ZagazPar_SepBlock[1, 2].adr2 := 1;
   ZagazPar_SepBlock[2, 1].adr1 := 12;
   ZagazPar_SepBlock[2, 1].adr2 := 2;
   ZagazPar_SepBlock[2, 2].adr1 := 12;
   ZagazPar_SepBlock[2, 2].adr2 := 3;
   ZagazPar_SepBlock[3, 1].adr1 := 12;
   ZagazPar_SepBlock[3, 1].adr2 := 4;
   ZagazPar_SepBlock[3, 2].adr1 := 12;
   ZagazPar_SepBlock[3, 2].adr2 := 5;
   ZagazPar_SepBlock[4, 1].adr1 := 12;
   ZagazPar_SepBlock[4, 1].adr2 := 6;
   ZagazPar_SepBlock[4, 2].adr1 := 12;
   ZagazPar_SepBlock[4, 2].adr2 := 7;
   ZagazPar_SepBlock[5, 1].adr1 := 13;
   ZagazPar_SepBlock[5, 1].adr2 := 1;
   ZagazPar_SepBlock[5, 2].adr1 := 13;
   ZagazPar_SepBlock[5, 2].adr2 := 2;
   ZagazPar_SepBlock[6, 1].adr1 := 13;
   ZagazPar_SepBlock[6, 1].adr2 := 3;
   ZagazPar_SepBlock[6, 2].adr1 := 13;
   ZagazPar_SepBlock[6, 2].adr2 := 4;
   ZagazPar_OperBlock[1, 1].adr1 := 13;
   ZagazPar_OperBlock[1, 1].adr2 := 6;
   ZagazPar_OperBlock[1, 2].adr1 := 13;
   ZagazPar_OperBlock[1, 2].adr2 := 7;
   ZagazPar_UouBlock[1, 1].adr1 := 9;
   ZagazPar_UouBlock[1, 2].adr1 := 9;
   ZagazPar_UouBlock[1, 2].adr2 := 1;
   ZagazPar_UouBlock[2, 1].adr1 := 9;
   ZagazPar_UouBlock[2, 1].adr2 := 2;
   ZagazPar_UouBlock[2, 2].adr1 := 9;
   ZagazPar_UouBlock[2, 2].adr2 := 3;
   ZagazPar_UouBlock[3, 1].adr1 := 9;
   ZagazPar_UouBlock[3, 1].adr2 := 4;
   ZagazPar_UouBlock[3, 2].adr1 := 9;
   ZagazPar_UouBlock[3, 2].adr2 := 5;
   ZagazPar_UouBlock[4, 1].adr1 := 9;
   ZagazPar_UouBlock[4, 1].adr2 := 6;
   ZagazPar_UouBlock[4, 2].adr1 := 9;
   ZagazPar_UouBlock[4, 2].adr2 := 7;
   ZagazPar_UouBlock[5, 1].adr1 := 10;
   ZagazPar_UouBlock[5, 2].adr1 := 10;
   ZagazPar_UouBlock[5, 2].adr2 := 1;
   ZagazPar_UouBlock[6, 1].adr1 := 10;
   ZagazPar_UouBlock[6, 1].adr2 := 2;
   ZagazPar_UouBlock[6, 2].adr1 := 10;
   ZagazPar_UouBlock[6, 2].adr2 := 3;
   ZagazPar_UouBlock[7, 1].adr1 := 10;
   ZagazPar_UouBlock[7, 1].adr2 := 4;
   ZagazPar_UouBlock[7, 2].adr1 := 10;
   ZagazPar_UouBlock[7, 2].adr2 := 5;
   ZagazPar_UouBlock[8, 1].adr1 := 10;
   ZagazPar_UouBlock[8, 1].adr2 := 6;
   ZagazPar_UouBlock[8, 2].adr1 := 10;
   ZagazPar_UouBlock[8, 2].adr2 := 7;
   ZagazPar_UouBlock[9, 1].adr1 := 11;
   ZagazPar_UouBlock[9, 2].adr1 := 11;
   ZagazPar_UouBlock[9, 2].adr2 := 1;
   ZagazPar_UouBlock[10, 1].adr1 := 11;
   ZagazPar_UouBlock[10, 1].adr2 := 2;
   ZagazPar_UouBlock[10, 2].adr1 := 11;
   ZagazPar_UouBlock[10, 2].adr2 := 3;
   ZagazPar_SepCHM10.adr1 := 13;
   ZagazPar_SepCHM10.adr2 := 5;
   ZagazPar_UouCHM10.adr1 := 11;
   ZagazPar_UouCHM10.adr2 := 4;
   PtnPar_HeaterOn.adr1 := 8;
   PtnPar_HeaterBreak.adr1 := 8;
   PtnPar_HeaterBreak.adr2 := 1;
   PtnPar_P_malo.adr1 := 8;
   PtnPar_P_malo.adr2 := 2;
   VsbPar_P_DoE1Malo.adr1 := 8;
   VsbPar_P_DoE1Malo.adr2 := 3;
   VsbPar_P_PosleE1Malo.adr1 := 8;
   VsbPar_P_PosleE1Malo.adr2 := 4;
   LitPar_T_ObrVodii_AvtVkl.adr1 := 14;
   LitPar_T_ObrVodii_AvtVkl.adr2 := 2;
   LitPar_ObogrevIT_Vkl.adr1 := 14;
   LitPar_ObogrevIT_Viikl.adr1 := 14;
   LitPar_ObogrevIT_Viikl.adr2 := 1;
   LitPar_ObogrevIT_Avariia.adr1 := 14;
   LitPar_ObogrevIT_Avariia.adr2 := 3;
   ZagazUpr_SepSignal_Svet1.adr1 := 4;
   ZagazUpr_SepSignal_Svet1.adr2 := 1;
   ZagazUpr_SepSignal_Svet2.adr1 := 4;
   ZagazUpr_SepSignal_Svet2.adr2 := 2;
   ZagazUpr_SepSignal_Zvuk1.adr1 := 4;
   ZagazUpr_SepSignal_Zvuk1.adr2 := 3;
   ZagazUpr_OperSignal_Svet.adr1 := 4;
   ZagazUpr_OperSignal_Svet.adr2 := 4;
   ZagazUpr_OperSignal_Zvuk.adr1 := 4;
   ZagazUpr_OperSignal_Zvuk.adr2 := 5;
   ZagazUpr_UouSignal_Svet.adr1 := 4;
END_DATA_BLOCK

DATA_BLOCK "DbSensAI"	// DB 223
TITLE = 'Значения параметров'
AUTHOR : Konst
FAMILY : Main
NAME : DbSensAI
VERSION : 0.0
  STRUCT
   numSensAIParam : INT ;
   SensAIParam : ARRAY  [0 .. 15 ] OF UDT 203;
  END_STRUCT ;	//Db
BEGIN
   numSensAIParam := 15;
   SensAIParam[0].adrPIW := 542;
   SensAIParam[0].BoundLoLo := 8.888880e+02;
   SensAIParam[0].BoundLo := 8.888880e+02;
   SensAIParam[0].BoundHi := 8.888880e+02;
   SensAIParam[0].BoundHiHi := 8.888880e+02;
   SensAIParam[0].HiMeasure := 1.000000e+02;
   SensAIParam[0].LoMeasure_mA := 4.000000e+00;
   SensAIParam[0].HiMeasure_mA := 2.000000e+01;
   SensAIParam[0].LoWorkRange_mA := 3.800000e+00;
   SensAIParam[0].HiWorkRange_mA := 2.020000e+01;
   SensAIParam[0].HmiSyncRange := 1;
   SensAIParam[1].adrPIW := 526;
   SensAIParam[1].BoundLoLo := 8.888880e+02;
   SensAIParam[1].BoundLo := 8.888880e+02;
   SensAIParam[1].BoundHi := 8.888880e+02;
   SensAIParam[1].BoundHiHi := 8.888880e+02;
   SensAIParam[1].LoMeasure := -5.000000e+01;
   SensAIParam[1].HiMeasure := 1.000000e+02;
   SensAIParam[1].LoMeasure_mA := 4.000000e+00;
   SensAIParam[1].HiMeasure_mA := 2.000000e+01;
   SensAIParam[1].LoWorkRange_mA := 3.800000e+00;
   SensAIParam[1].HiWorkRange_mA := 2.020000e+01;
   SensAIParam[1].HmiSyncRange := 1;
   SensAIParam[2].adrPIW := 524;
   SensAIParam[2].BoundLoLo := 8.888880e+02;
   SensAIParam[2].BoundLo := 8.888880e+02;
   SensAIParam[2].BoundHi := 8.888880e+02;
   SensAIParam[2].BoundHiHi := 8.888880e+02;
   SensAIParam[2].HiMeasure := 6.300000e+00;
   SensAIParam[2].LoMeasure_mA := 4.000000e+00;
   SensAIParam[2].HiMeasure_mA := 2.000000e+01;
   SensAIParam[2].LoWorkRange_mA := 3.800000e+00;
   SensAIParam[2].HiWorkRange_mA := 2.020000e+01;
   SensAIParam[2].HmiSyncRange := 1;
   SensAIParam[3].adrPIW := 528;
   SensAIParam[3].BoundLoLo := 8.888880e+02;
   SensAIParam[3].BoundLo := 8.888880e+02;
   SensAIParam[3].BoundHi := 8.888880e+02;
   SensAIParam[3].BoundHiHi := 8.888880e+02;
   SensAIParam[3].HiMeasure := 6.300000e+01;
   SensAIParam[3].LoMeasure_mA := 4.000000e+00;
   SensAIParam[3].HiMeasure_mA := 2.000000e+01;
   SensAIParam[3].LoWorkRange_mA := 3.800000e+00;
   SensAIParam[3].HiWorkRange_mA := 2.020000e+01;
   SensAIParam[3].HmiSyncRange := 1;
   SensAIParam[4].adrPIW := 530;
   SensAIParam[4].BoundLoLo := 8.888880e+02;
   SensAIParam[4].BoundLo := 8.888880e+02;
   SensAIParam[4].BoundHi := 8.888880e+02;
   SensAIParam[4].BoundHiHi := 8.888880e+02;
   SensAIParam[4].HiMeasure := 2.000000e+01;
   SensAIParam[4].LoMeasure_mA := 4.000000e+00;
   SensAIParam[4].HiMeasure_mA := 2.000000e+01;
   SensAIParam[4].LoWorkRange_mA := 3.800000e+00;
   SensAIParam[4].HiWorkRange_mA := 2.020000e+01;
   SensAIParam[4].HmiSyncRange := 1;
   SensAIParam[5].adrPIW := 522;
   SensAIParam[5].BoundLoLo := 3.000000e+01;
   SensAIParam[5].BoundLo := 3.500000e+01;
   SensAIParam[5].BoundHi := 5.200000e+01;
   SensAIParam[5].BoundHiHi := 5.500000e+01;
   SensAIParam[5].HiMeasure := 1.000000e+02;
   SensAIParam[5].LoMeasure_mA := 4.000000e+00;
   SensAIParam[5].HiMeasure_mA := 2.000000e+01;
   SensAIParam[5].LoWorkRange_mA := 3.800000e+00;
   SensAIParam[5].HiWorkRange_mA := 2.020000e+01;
   SensAIParam[5].HmiSyncRange := 1;
   SensAIParam[6].adrPIW := 536;
   SensAIParam[6].BoundLoLo := 8.888880e+02;
   SensAIParam[6].BoundLo := 8.888880e+02;
   SensAIParam[6].BoundHi := 8.888880e+02;
   SensAIParam[6].BoundHiHi := 8.888880e+02;
   SensAIParam[6].LoMeasure := -5.000000e+01;
   SensAIParam[6].HiMeasure := 1.000000e+02;
   SensAIParam[6].LoMeasure_mA := 4.000000e+00;
   SensAIParam[6].HiMeasure_mA := 2.000000e+01;
   SensAIParam[6].LoWorkRange_mA := 3.800000e+00;
   SensAIParam[6].HiWorkRange_mA := 2.020000e+01;
   SensAIParam[6].HmiSyncRange := 1;
   SensAIParam[7].adrPIW := 534;
   SensAIParam[7].BoundLoLo := 8.888880e+02;
   SensAIParam[7].BoundLo := 8.888880e+02;
   SensAIParam[7].BoundHi := 8.888880e+02;
   SensAIParam[7].BoundHiHi := 8.888880e+02;
   SensAIParam[7].HiMeasure := 6.300000e+00;
   SensAIParam[7].LoMeasure_mA := 4.000000e+00;
   SensAIParam[7].HiMeasure_mA := 2.000000e+01;
   SensAIParam[7].LoWorkRange_mA := 3.800000e+00;
   SensAIParam[7].HiWorkRange_mA := 2.020000e+01;
   SensAIParam[7].HmiSyncRange := 1;
   SensAIParam[8].adrPIW := 538;
   SensAIParam[8].BoundLoLo := 8.888880e+02;
   SensAIParam[8].BoundLo := 8.888880e+02;
   SensAIParam[8].BoundHi := 8.888880e+02;
   SensAIParam[8].BoundHiHi := 8.888880e+02;
   SensAIParam[8].HiMeasure := 6.300000e+01;
   SensAIParam[8].LoMeasure_mA := 4.000000e+00;
   SensAIParam[8].HiMeasure_mA := 2.000000e+01;
   SensAIParam[8].LoWorkRange_mA := 3.800000e+00;
   SensAIParam[8].HiWorkRange_mA := 2.020000e+01;
   SensAIParam[8].HmiSyncRange := 1;
   SensAIParam[9].adrPIW := 540;
   SensAIParam[9].BoundLoLo := 8.888880e+02;
   SensAIParam[9].BoundLo := 8.888880e+02;
   SensAIParam[9].BoundHi := 8.888880e+02;
   SensAIParam[9].BoundHiHi := 8.888880e+02;
   SensAIParam[9].HiMeasure := 2.000000e+01;
   SensAIParam[9].LoMeasure_mA := 4.000000e+00;
   SensAIParam[9].HiMeasure_mA := 2.000000e+01;
   SensAIParam[9].LoWorkRange_mA := 3.800000e+00;
   SensAIParam[9].HiWorkRange_mA := 2.020000e+01;
   SensAIParam[9].HmiSyncRange := 1;
   SensAIParam[10].adrPIW := 532;
   SensAIParam[10].BoundLoLo := 3.000000e+01;
   SensAIParam[10].BoundLo := 3.500000e+01;
   SensAIParam[10].BoundHi := 5.200000e+01;
   SensAIParam[10].BoundHiHi := 5.500000e+01;
   SensAIParam[10].HiMeasure := 1.000000e+02;
   SensAIParam[10].LoMeasure_mA := 4.000000e+00;
   SensAIParam[10].HiMeasure_mA := 2.000000e+01;
   SensAIParam[10].LoWorkRange_mA := 3.800000e+00;
   SensAIParam[10].HiWorkRange_mA := 2.020000e+01;
   SensAIParam[10].HmiSyncRange := 1;
   SensAIParam[11].adrPIW := 516;
   SensAIParam[11].BoundLoLo := 8.888880e+02;
   SensAIParam[11].BoundLo := 8.888880e+02;
   SensAIParam[11].BoundHi := 8.888880e+02;
   SensAIParam[11].BoundHiHi := 8.888880e+02;
   SensAIParam[11].LoMeasure := -5.000000e+01;
   SensAIParam[11].HiMeasure := 1.000000e+02;
   SensAIParam[11].LoMeasure_mA := 4.000000e+00;
   SensAIParam[11].HiMeasure_mA := 2.000000e+01;
   SensAIParam[11].LoWorkRange_mA := 3.800000e+00;
   SensAIParam[11].HiWorkRange_mA := 2.020000e+01;
   SensAIParam[11].HmiSyncRange := 1;
   SensAIParam[12].adrPIW := 514;
   SensAIParam[12].BoundLoLo := 8.888880e+02;
   SensAIParam[12].BoundLo := 8.888880e+02;
   SensAIParam[12].BoundHi := 8.888880e+02;
   SensAIParam[12].BoundHiHi := 8.888880e+02;
   SensAIParam[12].HiMeasure := 6.300000e+00;
   SensAIParam[12].LoMeasure_mA := 4.000000e+00;
   SensAIParam[12].HiMeasure_mA := 2.000000e+01;
   SensAIParam[12].LoWorkRange_mA := 3.800000e+00;
   SensAIParam[12].HiWorkRange_mA := 2.020000e+01;
   SensAIParam[12].HmiSyncRange := 1;
   SensAIParam[13].adrPIW := 518;
   SensAIParam[13].BoundLoLo := 8.888880e+02;
   SensAIParam[13].BoundLo := 8.888880e+02;
   SensAIParam[13].BoundHi := 8.888880e+02;
   SensAIParam[13].BoundHiHi := 8.888880e+02;
   SensAIParam[13].HiMeasure := 6.300000e+01;
   SensAIParam[13].LoMeasure_mA := 4.000000e+00;
   SensAIParam[13].HiMeasure_mA := 2.000000e+01;
   SensAIParam[13].LoWorkRange_mA := 3.800000e+00;
   SensAIParam[13].HiWorkRange_mA := 2.020000e+01;
   SensAIParam[13].HmiSyncRange := 1;
   SensAIParam[14].adrPIW := 520;
   SensAIParam[14].BoundLoLo := 8.888880e+02;
   SensAIParam[14].BoundLo := 8.888880e+02;
   SensAIParam[14].BoundHi := 8.888880e+02;
   SensAIParam[14].BoundHiHi := 8.888880e+02;
   SensAIParam[14].HiMeasure := 2.000000e+01;
   SensAIParam[14].LoMeasure_mA := 4.000000e+00;
   SensAIParam[14].HiMeasure_mA := 2.000000e+01;
   SensAIParam[14].LoWorkRange_mA := 3.800000e+00;
   SensAIParam[14].HiWorkRange_mA := 2.020000e+01;
   SensAIParam[14].HmiSyncRange := 1;
   SensAIParam[15].adrPIW := 512;
   SensAIParam[15].BoundLoLo := 3.000000e+01;
   SensAIParam[15].BoundLo := 3.500000e+01;
   SensAIParam[15].BoundHi := 5.200000e+01;
   SensAIParam[15].BoundHiHi := 5.500000e+01;
   SensAIParam[15].HiMeasure := 1.000000e+02;
   SensAIParam[15].LoMeasure_mA := 4.000000e+00;
   SensAIParam[15].HiMeasure_mA := 2.000000e+01;
   SensAIParam[15].LoWorkRange_mA := 3.800000e+00;
   SensAIParam[15].HiWorkRange_mA := 2.020000e+01;
   SensAIParam[15].HmiSyncRange := 1;
END_DATA_BLOCK

DATA_BLOCK "DbKranPpuAdr"	// DB 224
TITLE = 'Значения параметров'
AUTHOR : Konst
FAMILY : Main
NAME : DbKranP1
VERSION : 0.0
  STRUCT
   KranPpuEmul : BOOL ;	// эмуляция сигналов I,Q : 0 - выключена (реальные сигналы!) \ 1 - эмуляция
   SignalCopyToEmul : BOOL ;	// метка: 1- значения сигналов I[],Q[] копируются в виртуальные \ 0-нет
   KranPpuAdrParam : ARRAY  [1 .. 15, 1 .. 6 ] OF UDT 202;	//TAdrIOSignal;
  END_STRUCT ;	//Db
BEGIN
   KranPpuAdrParam[1, 1].adr1 := 4;
   KranPpuAdrParam[1, 2].adr1 := 4;
   KranPpuAdrParam[1, 2].adr2 := 1;
   KranPpuAdrParam[1, 3].adr1 := 5;
   KranPpuAdrParam[1, 3].adr2 := 1;
   KranPpuAdrParam[1, 4].adr1 := 5;
   KranPpuAdrParam[1, 4].adr2 := 2;
   KranPpuAdrParam[1, 5].adr1 := 2;
   KranPpuAdrParam[1, 6].adr1 := 2;
   KranPpuAdrParam[1, 6].adr2 := 1;
   KranPpuAdrParam[2, 1].adr1 := 4;
   KranPpuAdrParam[2, 1].adr2 := 2;
   KranPpuAdrParam[2, 2].adr1 := 4;
   KranPpuAdrParam[2, 2].adr2 := 3;
   KranPpuAdrParam[2, 3].adr1 := 5;
   KranPpuAdrParam[2, 3].adr2 := 3;
   KranPpuAdrParam[2, 4].adr1 := 5;
   KranPpuAdrParam[2, 4].adr2 := 4;
   KranPpuAdrParam[2, 5].adr1 := 2;
   KranPpuAdrParam[2, 5].adr2 := 2;
   KranPpuAdrParam[2, 6].adr1 := 2;
   KranPpuAdrParam[2, 6].adr2 := 3;
   KranPpuAdrParam[3, 1].adr1 := 4;
   KranPpuAdrParam[3, 1].adr2 := 6;
   KranPpuAdrParam[3, 2].adr1 := 4;
   KranPpuAdrParam[3, 2].adr2 := 7;
   KranPpuAdrParam[3, 3].adr1 := 5;
   KranPpuAdrParam[3, 3].adr2 := 7;
   KranPpuAdrParam[3, 4].adr1 := 5;
   KranPpuAdrParam[3, 5].adr1 := 2;
   KranPpuAdrParam[3, 5].adr2 := 6;
   KranPpuAdrParam[3, 6].adr1 := 2;
   KranPpuAdrParam[3, 6].adr2 := 7;
   KranPpuAdrParam[4, 1].adr1 := 4;
   KranPpuAdrParam[4, 1].adr2 := 4;
   KranPpuAdrParam[4, 2].adr1 := 4;
   KranPpuAdrParam[4, 2].adr2 := 5;
   KranPpuAdrParam[4, 3].adr1 := 5;
   KranPpuAdrParam[4, 3].adr2 := 5;
   KranPpuAdrParam[4, 4].adr1 := 5;
   KranPpuAdrParam[4, 4].adr2 := 6;
   KranPpuAdrParam[4, 5].adr1 := 2;
   KranPpuAdrParam[4, 5].adr2 := 4;
   KranPpuAdrParam[4, 6].adr1 := 2;
   KranPpuAdrParam[4, 6].adr2 := 5;
   KranPpuAdrParam[5, 1].adr1 := 6;
   KranPpuAdrParam[5, 1].adr2 := 4;
   KranPpuAdrParam[5, 2].adr1 := 6;
   KranPpuAdrParam[5, 2].adr2 := 5;
   KranPpuAdrParam[5, 3].adr1 := 7;
   KranPpuAdrParam[5, 3].adr2 := 3;
   KranPpuAdrParam[5, 4].adr1 := 7;
   KranPpuAdrParam[5, 4].adr2 := 4;
   KranPpuAdrParam[5, 5].adr1 := 3;
   KranPpuAdrParam[5, 5].adr2 := 4;
   KranPpuAdrParam[5, 6].adr1 := 3;
   KranPpuAdrParam[5, 6].adr2 := 5;
   KranPpuAdrParam[6, 1].adr1 := 6;
   KranPpuAdrParam[6, 1].adr2 := 2;
   KranPpuAdrParam[6, 2].adr1 := 6;
   KranPpuAdrParam[6, 2].adr2 := 3;
   KranPpuAdrParam[6, 3].adr1 := 7;
   KranPpuAdrParam[6, 3].adr2 := 1;
   KranPpuAdrParam[6, 4].adr1 := 7;
   KranPpuAdrParam[6, 4].adr2 := 2;
   KranPpuAdrParam[6, 5].adr1 := 3;
   KranPpuAdrParam[6, 5].adr2 := 2;
   KranPpuAdrParam[6, 6].adr1 := 3;
   KranPpuAdrParam[6, 6].adr2 := 3;
   KranPpuAdrParam[7, 1].adr1 := 6;
   KranPpuAdrParam[7, 1].adr2 := 6;
   KranPpuAdrParam[7, 2].adr1 := 6;
   KranPpuAdrParam[7, 2].adr2 := 7;
   KranPpuAdrParam[7, 3].adr1 := 7;
   KranPpuAdrParam[7, 3].adr2 := 5;
   KranPpuAdrParam[7, 4].adr1 := 7;
   KranPpuAdrParam[7, 4].adr2 := 6;
   KranPpuAdrParam[7, 5].adr1 := 3;
   KranPpuAdrParam[7, 5].adr2 := 6;
   KranPpuAdrParam[7, 6].adr1 := 3;
   KranPpuAdrParam[7, 6].adr2 := 7;
   KranPpuAdrParam[8, 1].adr1 := 6;
   KranPpuAdrParam[8, 2].adr1 := 6;
   KranPpuAdrParam[8, 2].adr2 := 1;
   KranPpuAdrParam[8, 3].adr1 := 7;
   KranPpuAdrParam[8, 3].adr2 := 7;
   KranPpuAdrParam[8, 4].adr1 := 7;
   KranPpuAdrParam[8, 5].adr1 := 3;
   KranPpuAdrParam[8, 6].adr1 := 3;
   KranPpuAdrParam[8, 6].adr2 := 1;
   KranPpuAdrParam[9, 2].adr2 := 1;
   KranPpuAdrParam[9, 3].adr1 := 1;
   KranPpuAdrParam[9, 3].adr2 := 7;
   KranPpuAdrParam[9, 4].adr1 := 1;
   KranPpuAdrParam[9, 6].adr2 := 1;
   KranPpuAdrParam[10, 1].adr2 := 2;
   KranPpuAdrParam[10, 2].adr2 := 3;
   KranPpuAdrParam[10, 3].adr1 := 2;
   KranPpuAdrParam[10, 4].adr1 := 2;
   KranPpuAdrParam[10, 4].adr2 := 1;
   KranPpuAdrParam[10, 5].adr2 := 2;
   KranPpuAdrParam[10, 6].adr2 := 3;
   KranPpuAdrParam[11, 1].adr2 := 6;
   KranPpuAdrParam[11, 2].adr2 := 7;
   KranPpuAdrParam[11, 3].adr1 := 2;
   KranPpuAdrParam[11, 3].adr2 := 4;
   KranPpuAdrParam[11, 4].adr1 := 2;
   KranPpuAdrParam[11, 4].adr2 := 5;
   KranPpuAdrParam[11, 5].adr2 := 6;
   KranPpuAdrParam[11, 6].adr2 := 7;
   KranPpuAdrParam[12, 1].adr2 := 4;
   KranPpuAdrParam[12, 2].adr2 := 5;
   KranPpuAdrParam[12, 3].adr1 := 2;
   KranPpuAdrParam[12, 3].adr2 := 2;
   KranPpuAdrParam[12, 4].adr1 := 2;
   KranPpuAdrParam[12, 4].adr2 := 3;
   KranPpuAdrParam[12, 5].adr2 := 4;
   KranPpuAdrParam[12, 6].adr2 := 5;
   KranPpuAdrParam[13, 1].adr1 := 1;
   KranPpuAdrParam[13, 1].adr2 := 3;
   KranPpuAdrParam[13, 2].adr1 := 1;
   KranPpuAdrParam[13, 2].adr2 := 4;
   KranPpuAdrParam[13, 3].adr1 := 3;
   KranPpuAdrParam[13, 4].adr1 := 3;
   KranPpuAdrParam[13, 4].adr2 := 1;
   KranPpuAdrParam[13, 5].adr1 := 1;
   KranPpuAdrParam[13, 5].adr2 := 2;
   KranPpuAdrParam[13, 6].adr1 := 1;
   KranPpuAdrParam[13, 6].adr2 := 3;
   KranPpuAdrParam[14, 1].adr1 := 1;
   KranPpuAdrParam[14, 1].adr2 := 1;
   KranPpuAdrParam[14, 2].adr1 := 1;
   KranPpuAdrParam[14, 2].adr2 := 2;
   KranPpuAdrParam[14, 3].adr1 := 2;
   KranPpuAdrParam[14, 3].adr2 := 6;
   KranPpuAdrParam[14, 4].adr1 := 2;
   KranPpuAdrParam[14, 4].adr2 := 7;
   KranPpuAdrParam[14, 5].adr1 := 1;
   KranPpuAdrParam[14, 6].adr1 := 1;
   KranPpuAdrParam[14, 6].adr2 := 1;
   KranPpuAdrParam[15, 1].adr1 := 1;
   KranPpuAdrParam[15, 1].adr2 := 5;
   KranPpuAdrParam[15, 2].adr1 := 1;
   KranPpuAdrParam[15, 2].adr2 := 6;
   KranPpuAdrParam[15, 3].adr1 := 3;
   KranPpuAdrParam[15, 3].adr2 := 2;
   KranPpuAdrParam[15, 4].adr1 := 3;
   KranPpuAdrParam[15, 4].adr2 := 3;
   KranPpuAdrParam[15, 5].adr1 := 1;
   KranPpuAdrParam[15, 5].adr2 := 4;
   KranPpuAdrParam[15, 6].adr1 := 1;
   KranPpuAdrParam[15, 6].adr2 := 5;
END_DATA_BLOCK

DATA_BLOCK "DbKranPpu"	// DB 225
TITLE = 'Значения параметров'
AUTHOR : Konst
FAMILY : Main
NAME : DbKranP2
VERSION : 0.0
  STRUCT
   numKrPpu : INT ;	// количество кранов ЭППУ
   SignalCloseOff : BOOL ;	//метка: 1- выключить Выходные сигналы для всех кранов\ 0-нет
   SignalOpenOff : BOOL ;	//метка: 1- выключить Входные сигналы для всех кранов\ 0-нет
   HandPushOff : BOOL ;	//метка: 1 - выкл. "HandPush" со снятием упр. сигналов для всех кранов\ 0-нет
   KranPpuParam : ARRAY  [1 .. 15 ] OF UDT 204;	// м. еще размерность или KranPpuParam_Prev
  END_STRUCT ;	//Db
BEGIN
   numKrPpu := 15;
   KranPpuParam[1].TmOperKr_NO := 101;
   KranPpuParam[1].TmStrag_Value := S5T#5S;
   KranPpuParam[1].TmFullClose_Value := S5T#20S;
   KranPpuParam[1].TmFullOpen_Value := S5T#20S;
   KranPpuParam[1].TmDogim_Value := S5T#3S;
   KranPpuParam[1].HmiSyncTimers := 1;
   KranPpuParam[2].TmOperKr_NO := 102;
   KranPpuParam[2].TmStrag_Value := S5T#5S;
   KranPpuParam[2].TmFullClose_Value := S5T#20S;
   KranPpuParam[2].TmFullOpen_Value := S5T#20S;
   KranPpuParam[2].TmDogim_Value := S5T#3S;
   KranPpuParam[2].HmiSyncTimers := 1;
   KranPpuParam[3].TmOperKr_NO := 103;
   KranPpuParam[3].TmStrag_Value := S5T#5S;
   KranPpuParam[3].TmFullClose_Value := S5T#20S;
   KranPpuParam[3].TmFullOpen_Value := S5T#20S;
   KranPpuParam[3].TmDogim_Value := S5T#3S;
   KranPpuParam[3].HmiSyncTimers := 1;
   KranPpuParam[4].TmOperKr_NO := 104;
   KranPpuParam[4].TmStrag_Value := S5T#5S;
   KranPpuParam[4].TmFullClose_Value := S5T#20S;
   KranPpuParam[4].TmFullOpen_Value := S5T#20S;
   KranPpuParam[4].TmDogim_Value := S5T#3S;
   KranPpuParam[4].HmiSyncTimers := 1;
   KranPpuParam[5].TmOperKr_NO := 105;
   KranPpuParam[5].TmStrag_Value := S5T#5S;
   KranPpuParam[5].TmFullClose_Value := S5T#20S;
   KranPpuParam[5].TmFullOpen_Value := S5T#20S;
   KranPpuParam[5].TmDogim_Value := S5T#3S;
   KranPpuParam[5].HmiSyncTimers := 1;
   KranPpuParam[6].TmOperKr_NO := 106;
   KranPpuParam[6].TmStrag_Value := S5T#5S;
   KranPpuParam[6].TmFullClose_Value := S5T#20S;
   KranPpuParam[6].TmFullOpen_Value := S5T#20S;
   KranPpuParam[6].TmDogim_Value := S5T#3S;
   KranPpuParam[6].HmiSyncTimers := 1;
   KranPpuParam[7].TmOperKr_NO := 107;
   KranPpuParam[7].TmStrag_Value := S5T#5S;
   KranPpuParam[7].TmFullClose_Value := S5T#20S;
   KranPpuParam[7].TmFullOpen_Value := S5T#20S;
   KranPpuParam[7].TmDogim_Value := S5T#3S;
   KranPpuParam[7].HmiSyncTimers := 1;
   KranPpuParam[8].TmOperKr_NO := 108;
   KranPpuParam[8].TmStrag_Value := S5T#5S;
   KranPpuParam[8].TmFullClose_Value := S5T#20S;
   KranPpuParam[8].TmFullOpen_Value := S5T#20S;
   KranPpuParam[8].TmDogim_Value := S5T#3S;
   KranPpuParam[8].HmiSyncTimers := 1;
   KranPpuParam[9].TmOperKr_NO := 109;
   KranPpuParam[9].TmStrag_Value := S5T#5S;
   KranPpuParam[9].TmFullClose_Value := S5T#20S;
   KranPpuParam[9].TmFullOpen_Value := S5T#20S;
   KranPpuParam[9].TmDogim_Value := S5T#3S;
   KranPpuParam[9].HmiSyncTimers := 1;
   KranPpuParam[10].TmOperKr_NO := 110;
   KranPpuParam[10].TmStrag_Value := S5T#5S;
   KranPpuParam[10].TmFullClose_Value := S5T#20S;
   KranPpuParam[10].TmFullOpen_Value := S5T#20S;
   KranPpuParam[10].TmDogim_Value := S5T#3S;
   KranPpuParam[10].HmiSyncTimers := 1;
   KranPpuParam[11].TmOperKr_NO := 111;
   KranPpuParam[11].TmStrag_Value := S5T#5S;
   KranPpuParam[11].TmFullClose_Value := S5T#20S;
   KranPpuParam[11].TmFullOpen_Value := S5T#20S;
   KranPpuParam[11].TmDogim_Value := S5T#3S;
   KranPpuParam[11].HmiSyncTimers := 1;
   KranPpuParam[12].TmOperKr_NO := 112;
   KranPpuParam[12].TmStrag_Value := S5T#5S;
   KranPpuParam[12].TmFullClose_Value := S5T#20S;
   KranPpuParam[12].TmFullOpen_Value := S5T#20S;
   KranPpuParam[12].TmDogim_Value := S5T#3S;
   KranPpuParam[12].HmiSyncTimers := 1;
   KranPpuParam[13].TmOperKr_NO := 113;
   KranPpuParam[13].TmStrag_Value := S5T#5S;
   KranPpuParam[13].TmFullClose_Value := S5T#20S;
   KranPpuParam[13].TmFullOpen_Value := S5T#20S;
   KranPpuParam[13].TmDogim_Value := S5T#3S;
   KranPpuParam[13].HmiSyncTimers := 1;
   KranPpuParam[14].TmOperKr_NO := 114;
   KranPpuParam[14].TmStrag_Value := S5T#5S;
   KranPpuParam[14].TmFullClose_Value := S5T#20S;
   KranPpuParam[14].TmFullOpen_Value := S5T#20S;
   KranPpuParam[14].TmDogim_Value := S5T#3S;
   KranPpuParam[14].HmiSyncTimers := 1;
   KranPpuParam[15].TmOperKr_NO := 115;
   KranPpuParam[15].TmStrag_Value := S5T#5S;
   KranPpuParam[15].TmFullClose_Value := S5T#20S;
   KranPpuParam[15].TmFullOpen_Value := S5T#20S;
   KranPpuParam[15].TmDogim_Value := S5T#3S;
   KranPpuParam[15].HmiSyncTimers := 1;
END_DATA_BLOCK

DATA_BLOCK "DbSepBu"	// DB 226
TITLE = 'Значения параметров БУ ВН2012'
AUTHOR : Konst
FAMILY : Main
NAME : DbSepBu
VERSION : 0.0
  STRUCT
   numSepBuParam : INT ;
   SepBuParam : ARRAY  [1 .. 4 ] OF UDT 206;
  END_STRUCT ;	//Db
BEGIN
   numSepBuParam := 4;
   SepBuParam[1].lblCopyErrToInvalid := TRUE;
   SepBuParam[2].lblCopyErrToInvalid := TRUE;
   SepBuParam[3].lblCopyErrToInvalid := TRUE;
   SepBuParam[4].lblCopyErrToInvalid := TRUE;
END_DATA_BLOCK

DATA_BLOCK "DbSipValve"	// DB 227
VERSION : 0.0
  STRUCT
   numSipValve : INT ;	// количество клапанов
   SipValveParam : ARRAY  [1 .. 5 ] OF UDT 207;
  END_STRUCT ;	//Db
BEGIN
   numSipValve := 5;
   SipValveParam[1].AddrPQW := 514;
   SipValveParam[1].ControlModeAuto := TRUE;
   SipValveParam[1].Value_Task_Percent := 100;
   SipValveParam[2].AddrPQW := 516;
   SipValveParam[2].ControlModeAuto := TRUE;
   SipValveParam[2].Value_Task_Percent := 100;
   SipValveParam[3].AddrPQW := 512;
   SipValveParam[3].ControlModeAuto := TRUE;
   SipValveParam[3].Value_Task_Percent := 100;
   SipValveParam[4].AddrPQW := 520;
   SipValveParam[4].ControlModeAuto := TRUE;
   SipValveParam[4].Value_Task_Percent := 100;
   SipValveParam[5].AddrPQW := 518;
   SipValveParam[5].ControlModeAuto := TRUE;
   SipValveParam[5].Value_Task_Percent := 100;
END_DATA_BLOCK

DATA_BLOCK "DbFlowData"	// DB 228
TITLE = 'Значения параметров БУ ВН2012'
AUTHOR : Konst
FAMILY : Main
NAME : DbCalc
VERSION : 0.0
  STRUCT
   numFlowData : INT ;	//количество элементов FlowData[]
   FlowData : ARRAY  [0 .. 7 ] OF UDT 208;
  END_STRUCT ;	//Db
BEGIN
   numFlowData := 7;
END_DATA_BLOCK

DATA_BLOCK "DbBitMess"	// DB 229
TITLE = 'Сообщения'
AUTHOR : Konst
FAMILY : Main
NAME : DbMess
VERSION : 0.0
  STRUCT
   Mess_AI_LoLo : WORD ;	//биты для сообщений о нарушение НАГ для датчииков AI, тип А\К (Авар\Красный)
   Mess_AI_Lo : WORD ;	//биты для сообщений о нарушение НПГ для датчииков AI, тип А\Ж (Авар\Желтый)
   Mess_AI_Hi : WORD ;	//биты для сообщений о нарушение ВПГ для датчииков AI, тип А\Ж
   Mess_AI_HiHi : WORD ;	//биты для сообщений о нарушение ВАГ для датчииков AI, тип А.К.(Андрей Конст)
   Mess_KrPpu_Close : WORD ;	//биты для сообщений об закрытии кранов , тип Инф
   Mess_KrPpu_Open : WORD ;	//биты для сообщений об открытии кранов , тип Инф
   Mess_KrPpu_ErrClose : WORD ;	//биты для сообщений об ошибке при закрытии кранов , тип А\Ж
   Mess_KrPpu_ErrOpen : WORD ;	//биты для сообщений об открытии кранов , тип А\Ж (Авар\Желтый)
   Mess_KrPpu_ErrFatal : WORD ;	//биты для сообщений о фатальной неиспр. кранов , тип А\К
   Mess_BU_ErrRefresh : WORD ;	//биты для сообщений об ошибке обновления данных с БУ(Нет сязи),тип А\Ж
   Mess_BU_Norm : WORD ;	//биты для сообщений о восстановлении связи с БУ,тип Инф
   Mess_AI_Norm : WORD ;	//биты для сообщений о зозврате значения датчика в норму,тип Инф
   Mess_KrPpu_Norm : WORD ;	//биты для сообщений о восстановлении исправности крана,тип Инф
  END_STRUCT ;	//Db
BEGIN
END_DATA_BLOCK

DATA_BLOCK "DbControl"	// DB 230
TITLE = 'Управление'
AUTHOR : Konst
FAMILY : Main
NAME : DbContr
VERSION : 0.0
  STRUCT
   DtSync_Hmi : UDT 210;	//int-компоненты даты для синхронизации времени Hmi=>Plc
   DtSync_Once : UDT 210;	//int-компоненты даты для дополнительного задания времени Plc
   lblDtSync_Hmi : BOOL ;	//метка о синхронизации DtPlc с Hmi : 1-синхронизировать\0-нет
   lblDtSync_Hmi_Ignore : BOOL ;	//метка об игнорировании синхронизации DtPlc с Hmi : 1-игнорировать\0-нет
   lblDtSync_Once : BOOL ;	//метка о доп-й синхронизации DtPlc через DtSync_Once: 1-синхронизировать\0-нет
   DtPlc_Change_Event : INT ;	//флаг события "изменение DtPlc":0-не изм.\1-ч/з DtSync_HMI\2-ч/з DtSync_Once
   DtPlc_Change_Counter : INT ;	//счётчик числа изменений DtPlc времени ПЛК ([1-30000])
   DtPlc_Change_Value_Time : TIME ;	//время в формате "Time", на которую изменилось DtPlc после синхронизации
   DtPlc_Change_Value_MSec : DINT ;	//время в мСек, на которую изменилось DtPlc после синхронизации
   DtPlc_Format_Int : UDT 210;	//время ПЛК DtPlc в формате int-компоненты даты
   DtPlc_Format_Str : STRING  [22 ];	//время ПЛК DtPlc в строковом формате "DD.MM.YY HH:MM:SS"
   FlowTG_Sens_Correct_Cut : REAL ;	//!!"отсечка" dX показания датчика РТГ (при V<dX, принимается V=0)
   FlowTG_Sens_Correct_0 : REAL ;	//!!"смещение нуля" dY показания датчика РТГ (при V>dX, принимается V=V-dY)
   isMode_AvOst : BOOL ;	//флаг активности события "Режим Аварийный Останов" для всей УПС: 0- нет\1- да
   isMode_AvOst_Prev : BOOL ;	//флаг события "Режим Аварийный Останов" - предыдущее значение
   isMode_RegimRemont : BOOL ;	//флаг активности события "Режим Ремонт" для всей подс-мы УПС: 0- нет\1- да
   isMode_RegimRemont_Prev : BOOL ;	//флаг события "Режим Ремонт" - предыдущее значение
  END_STRUCT ;	//Db
BEGIN
   DtSync_Hmi.Year := 2012;
   DtSync_Hmi.Month := 3;
   DtSync_Hmi.Day := 23;
   DtSync_Hmi.Hour := 17;
   DtSync_Hmi.Minute := 41;
   DtSync_Hmi.Sec := 27;
   DtSync_Hmi.MSec := 345;
   FlowTG_Sens_Correct_Cut := 5.000000e-02;
   FlowTG_Sens_Correct_0 := 3.000000e-02;
END_DATA_BLOCK

